// Mitsubishi GX Works2 project: InnerDrumTurnP202201050806   PLC: Q03UDV

PROGRAM MAIN
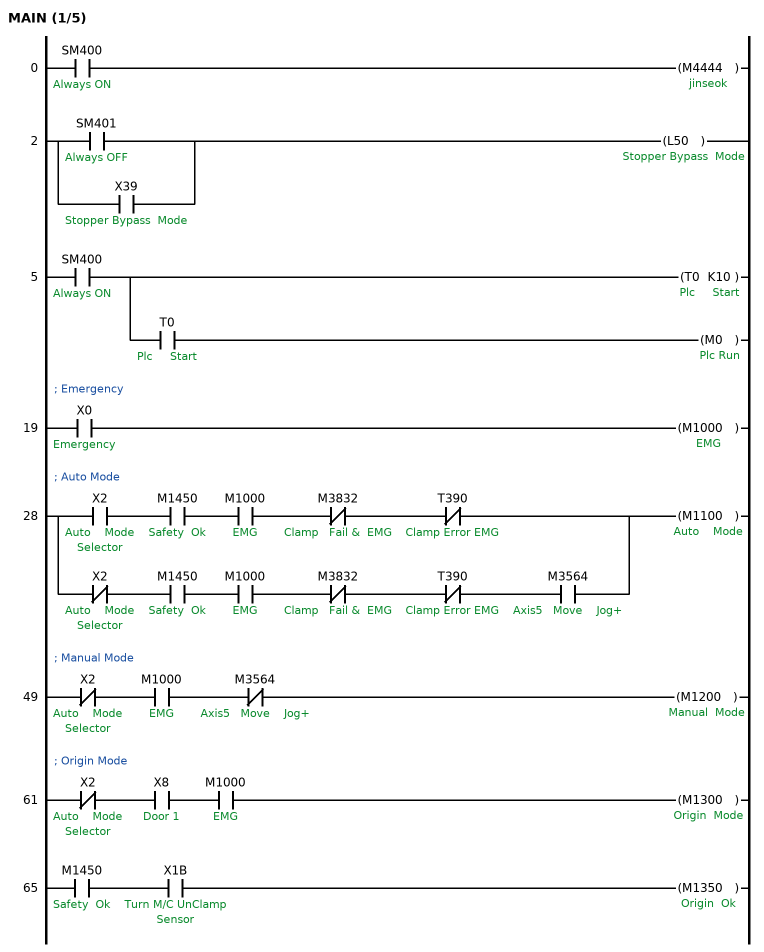
0     LD      SM400  ; Always ON
      OUT     M4444  ; jinseok
2     LD      SM401  ; Always OFF
      OR      X39  ; Stopper Bypass  Mode
      OUT     L50  ; Stopper Bypass  Mode
5     LD      SM400  ; Always ON
      OUT     T0 K10  ; Plc     Start
      AND     T0  ; Plc     Start
      OUT     M0  ; Plc Run
; Emergency
19    LD      X0  ; Emergency
      OUT     M1000  ; EMG
; Auto Mode
28    LD      X2  ; Auto    Mode    Selector
      AND     M1450  ; Safety  Ok
      AND     M1000  ; EMG
      ANI     M3832  ; Clamp   Fail &  EMG
      ANI     T390  ; Clamp Error EMG
      LDI     X2  ; Auto    Mode    Selector
      AND     M1450  ; Safety  Ok
      AND     M1000  ; EMG
      ANI     M3832  ; Clamp   Fail &  EMG
      ANI     T390  ; Clamp Error EMG
      AND     M3564  ; Axis5   Move    Jog+
      ORB
      OUT     M1100  ; Auto    Mode
; Manual Mode
49    LDI     X2  ; Auto    Mode    Selector
      AND     M1000  ; EMG
      ANI     M3564  ; Axis5   Move    Jog+
      OUT     M1200  ; Manual  Mode
; Origin Mode
61    LDI     X2  ; Auto    Mode    Selector
      AND     X8  ; Door 1
      AND     M1000  ; EMG
      OUT     M1300  ; Origin  Mode
65    LD      M1450  ; Safety  Ok
      AND     X1B  ; Turn M/C UnClamp Sensor
      OUT     M1350  ; Origin  Ok
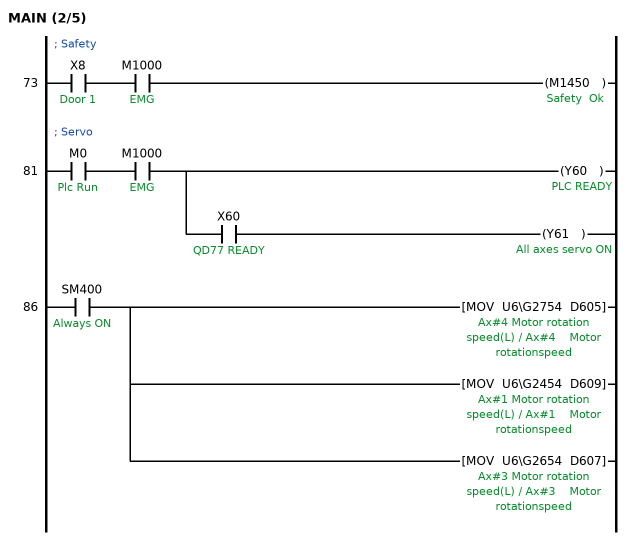
; Safety
73    LD      X8  ; Door 1
      AND     M1000  ; EMG
      OUT     M1450  ; Safety  Ok
; Servo
81    LD      M0  ; Plc Run
      AND     M1000  ; EMG
      OUT     Y60  ; PLC READY
      AND     X60  ; QD77 READY
      OUT     Y61  ; All axes servo ON
86    LD      SM400  ; Always ON
      MOV     U6\G2754 D605  ; Ax#4 Motor rotation speed(L) / Ax#4    Motor   rotationspeed
      MOV     U6\G2454 D609  ; Ax#1 Motor rotation speed(L) / Ax#1    Motor   rotationspeed
      MOV     U6\G2654 D607  ; Ax#3 Motor rotation speed(L) / Ax#3    Motor   rotationspeed
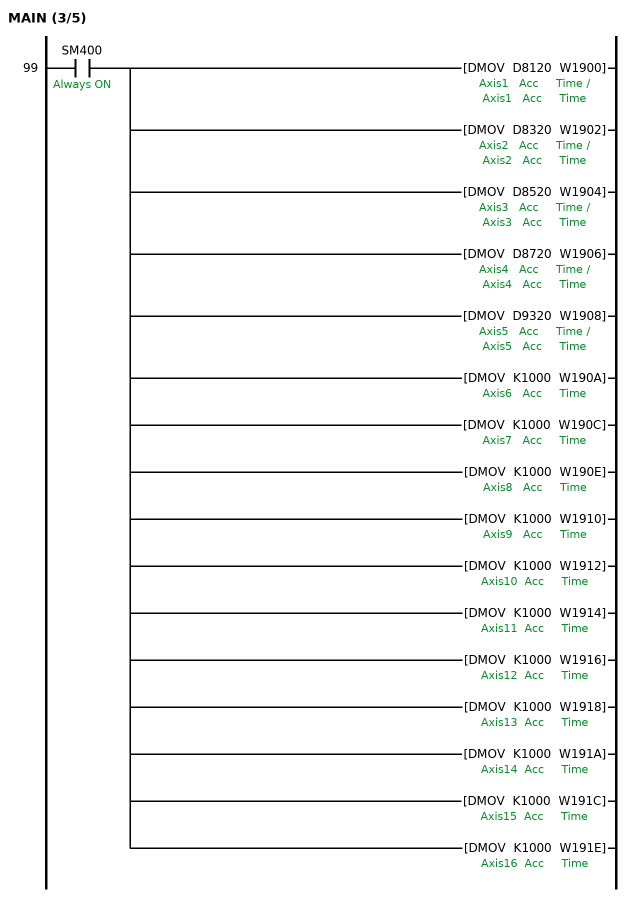
99    LD      SM400  ; Always ON
      DMOV    D8120 W1900  ; Axis1   Acc     Time / Axis1   Acc     Time
      DMOV    D8320 W1902  ; Axis2   Acc     Time / Axis2   Acc     Time
      DMOV    D8520 W1904  ; Axis3   Acc     Time / Axis3   Acc     Time
      DMOV    D8720 W1906  ; Axis4   Acc     Time / Axis4   Acc     Time
      DMOV    D9320 W1908  ; Axis5   Acc     Time / Axis5   Acc     Time
      DMOV    K1000 W190A  ; Axis6   Acc     Time
      DMOV    K1000 W190C  ; Axis7   Acc     Time
      DMOV    K1000 W190E  ; Axis8   Acc     Time
      DMOV    K1000 W1910  ; Axis9   Acc     Time
      DMOV    K1000 W1912  ; Axis10  Acc     Time
      DMOV    K1000 W1914  ; Axis11  Acc     Time
      DMOV    K1000 W1916  ; Axis12  Acc     Time
      DMOV    K1000 W1918  ; Axis13  Acc     Time
      DMOV    K1000 W191A  ; Axis14  Acc     Time
      DMOV    K1000 W191C  ; Axis15  Acc     Time
      DMOV    K1000 W191E  ; Axis16  Acc     Time
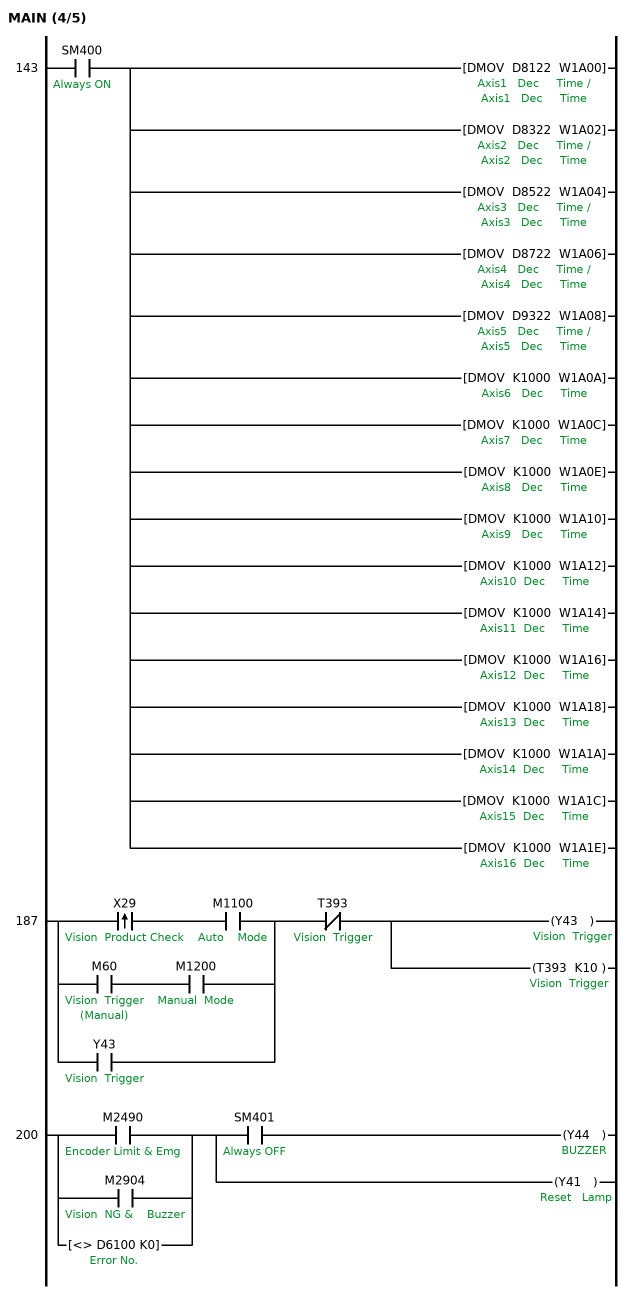
143   LD      SM400  ; Always ON
      DMOV    D8122 W1A00  ; Axis1   Dec     Time / Axis1   Dec     Time
      DMOV    D8322 W1A02  ; Axis2   Dec     Time / Axis2   Dec     Time
      DMOV    D8522 W1A04  ; Axis3   Dec     Time / Axis3   Dec     Time
      DMOV    D8722 W1A06  ; Axis4   Dec     Time / Axis4   Dec     Time
      DMOV    D9322 W1A08  ; Axis5   Dec     Time / Axis5   Dec     Time
      DMOV    K1000 W1A0A  ; Axis6   Dec     Time
      DMOV    K1000 W1A0C  ; Axis7   Dec     Time
      DMOV    K1000 W1A0E  ; Axis8   Dec     Time
      DMOV    K1000 W1A10  ; Axis9   Dec     Time
      DMOV    K1000 W1A12  ; Axis10  Dec     Time
      DMOV    K1000 W1A14  ; Axis11  Dec     Time
      DMOV    K1000 W1A16  ; Axis12  Dec     Time
      DMOV    K1000 W1A18  ; Axis13  Dec     Time
      DMOV    K1000 W1A1A  ; Axis14  Dec     Time
      DMOV    K1000 W1A1C  ; Axis15  Dec     Time
      DMOV    K1000 W1A1E  ; Axis16  Dec     Time
187   LDP     X29  ; Vision  Product Check
      AND     M1100  ; Auto    Mode
      LD      M60  ; Vision  Trigger (Manual)
      AND     M1200  ; Manual  Mode
      ORB
      OR      Y43  ; Vision  Trigger
      ANI     T393  ; Vision  Trigger
      OUT     Y43  ; Vision  Trigger
      OUT     T393 K10  ; Vision  Trigger
200   LD      M2490  ; Encoder Limit & Emg
      OR      M2904  ; Vision  NG &    Buzzer
      OR<>    D6100 K0  ; Error No.
      MPS
      AND     SM401  ; Always OFF
      OUT     Y44  ; BUZZER
      MPP
      OUT     Y41  ; Reset   Lamp
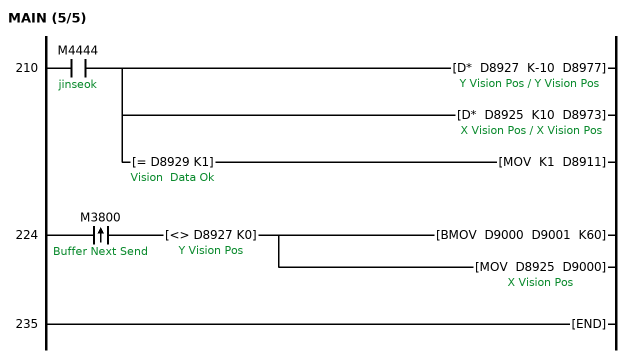
210   LD      M4444  ; jinseok
      D*      D8927 K-10 D8977  ; Y Vision Pos / Y Vision Pos
      D*      D8925 K10 D8973  ; X Vision Pos / X Vision Pos
      AND=    D8929 K1  ; Vision  Data Ok
      MOV     K1 D8911
224   LDP     M3800  ; Buffer Next Send
      AND<>   D8927 K0  ; Y Vision Pos
      BMOV    D9000 D9001 K60
      MOV     D8925 D9000
235   END
END_PROGRAM

PROGRAM AUTO
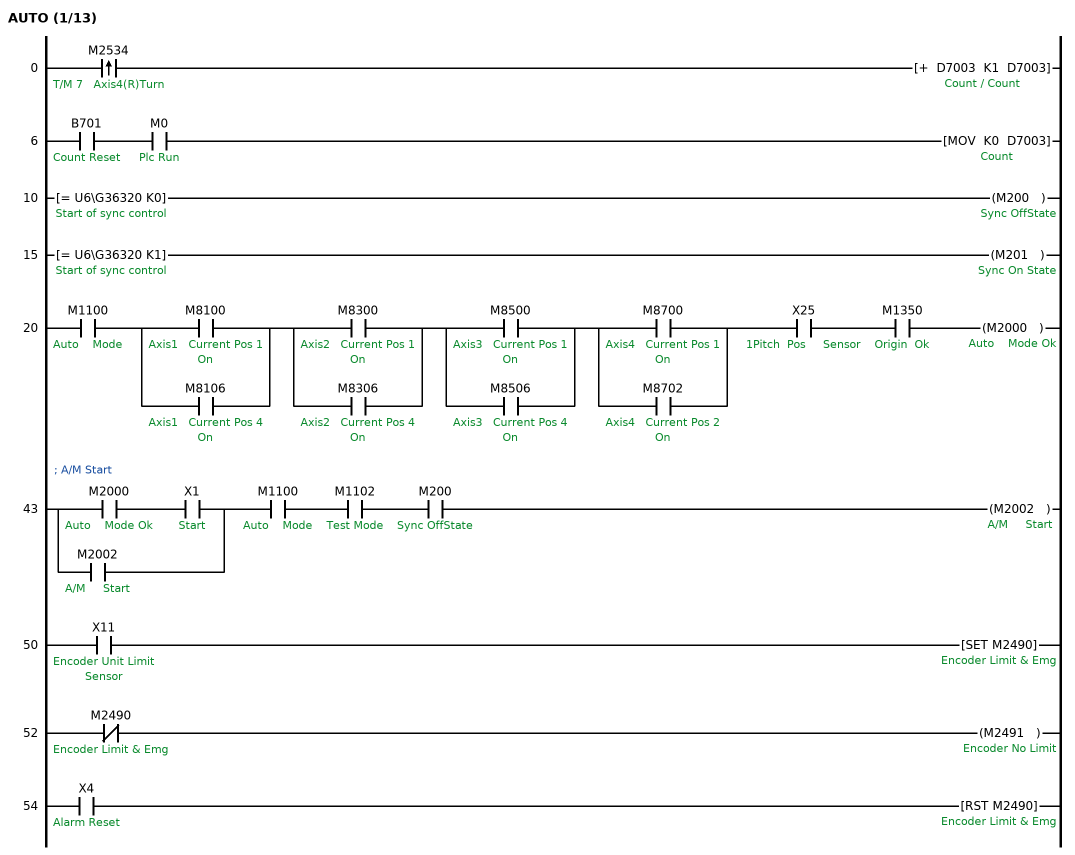
0     LDP     M2534  ; T/M 7   Axis4(R)Turn
      +       D7003 K1 D7003  ; Count
6     LD      B701  ; Count Reset
      AND     M0  ; Plc Run
      MOV     K0 D7003
10    LD=     U6\G36320 K0  ; Start of sync control
      OUT     M200  ; Sync OffState
15    LD=     U6\G36320 K1  ; Start of sync control
      OUT     M201  ; Sync On State
20    LD      M1100  ; Auto    Mode
      LD      M8100  ; Axis1   Current Pos 1 On
      OR      M8106  ; Axis1   Current Pos 4 On
      ANB
      LD      M8300  ; Axis2   Current Pos 1 On
      OR      M8306  ; Axis2   Current Pos 4 On
      ANB
      LD      M8500  ; Axis3   Current Pos 1 On
      OR      M8506  ; Axis3   Current Pos 4 On
      ANB
      LD      M8700  ; Axis4   Current Pos 1 On
      OR      M8702  ; Axis4   Current Pos 2 On
      ANB
      AND     X25  ; 1Pitch  Pos     Sensor
      AND     M1350  ; Origin  Ok
      OUT     M2000  ; Auto    Mode Ok
; A/M Start
43    LD      M2000  ; Auto    Mode Ok
      AND     X1  ; Start
      OR      M2002  ; A/M     Start
      AND     M1100  ; Auto    Mode
      AND     M1102  ; Test Mode
      AND     M200  ; Sync OffState
      OUT     M2002  ; A/M     Start
50    LD      X11  ; Encoder Unit Limit Sensor
      SET     M2490  ; Encoder Limit & Emg
52    LDI     M2490  ; Encoder Limit & Emg
      OUT     M2491  ; Encoder No Limit
54    LD      X4  ; Alarm Reset
      RST     M2490  ; Encoder Limit & Emg
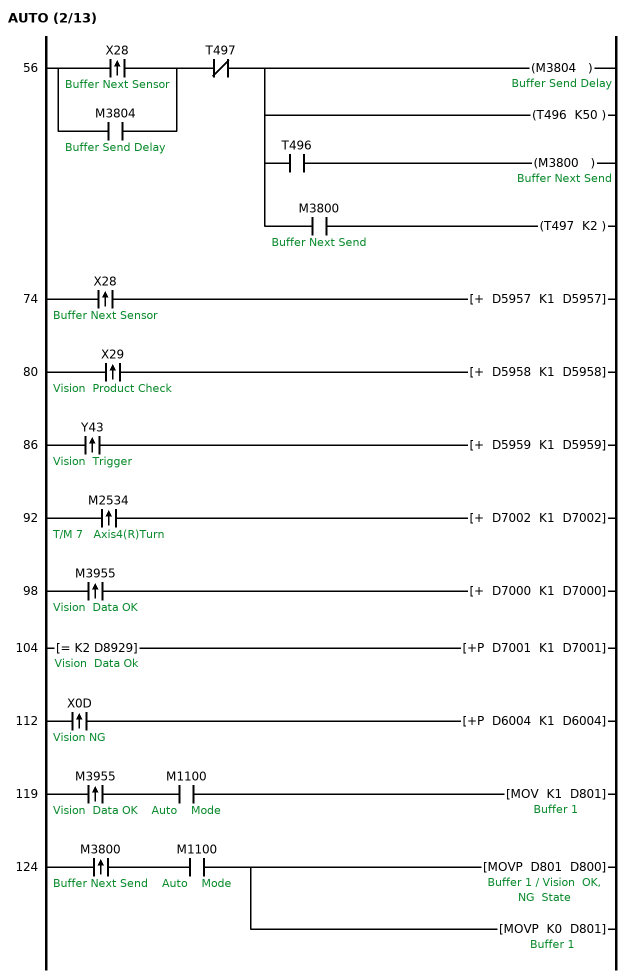
56    LDP     X28  ; Buffer Next Sensor
      OR      M3804  ; Buffer Send Delay
      ANI     T497
      OUT     M3804  ; Buffer Send Delay
      OUT     T496 K50
      MPS
      AND     T496
      OUT     M3800  ; Buffer Next Send
      MPP
      AND     M3800  ; Buffer Next Send
      OUT     T497 K2
74    LDP     X28  ; Buffer Next Sensor
      +       D5957 K1 D5957
80    LDP     X29  ; Vision  Product Check
      +       D5958 K1 D5958
86    LDP     Y43  ; Vision  Trigger
      +       D5959 K1 D5959
92    LDP     M2534  ; T/M 7   Axis4(R)Turn
      +       D7002 K1 D7002
98    LDP     M3955  ; Vision  Data OK
      +       D7000 K1 D7000
104   LD=     K2 D8929  ; Vision  Data Ok
      +P      D7001 K1 D7001
112   LDP     X0D  ; Vision NG
      +P      D6004 K1 D6004
119   LDP     M3955  ; Vision  Data OK
      AND     M1100  ; Auto    Mode
      MOV     K1 D801  ; Buffer 1
124   LDP     M3800  ; Buffer Next Send
      AND     M1100  ; Auto    Mode
      MOVP    D801 D800  ; Vision  OK, NG  State
      MOVP    K0 D801
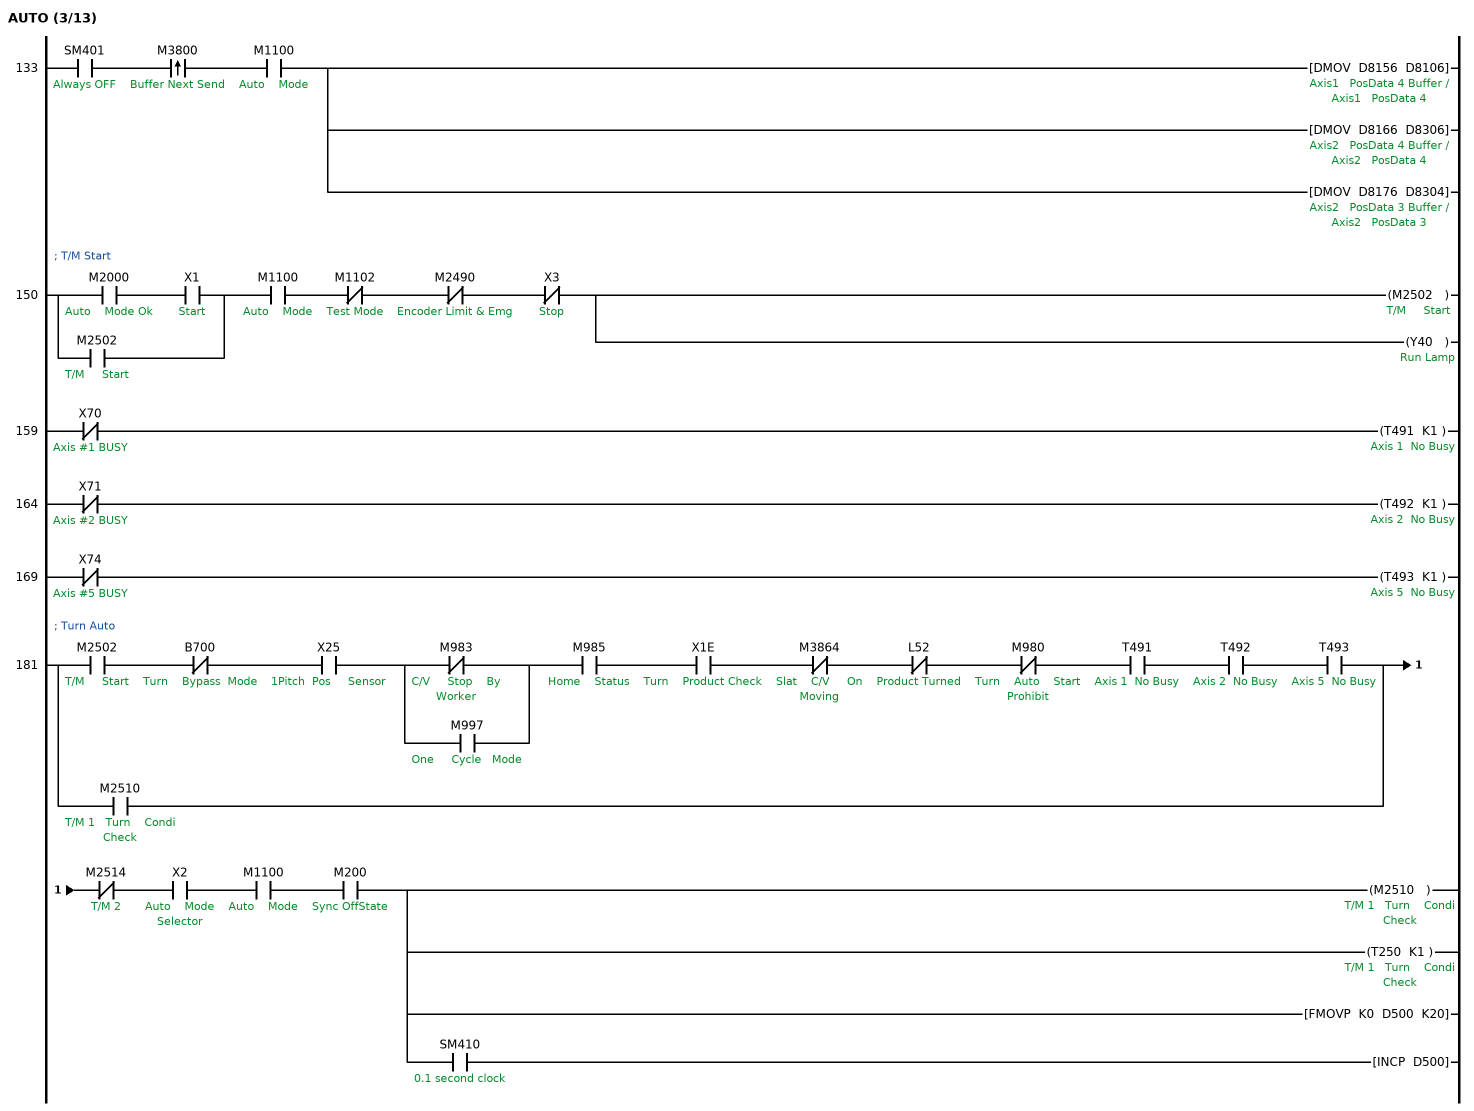
133   LD      SM401  ; Always OFF
      ANDP    M3800  ; Buffer Next Send
      AND     M1100  ; Auto    Mode
      DMOV    D8156 D8106  ; Axis1   PosData 4 Buffer / Axis1   PosData 4
      DMOV    D8166 D8306  ; Axis2   PosData 4 Buffer / Axis2   PosData 4
      DMOV    D8176 D8304  ; Axis2   PosData 3 Buffer / Axis2   PosData 3
; T/M Start
150   LD      M2000  ; Auto    Mode Ok
      AND     X1  ; Start
      OR      M2502  ; T/M     Start
      AND     M1100  ; Auto    Mode
      ANI     M1102  ; Test Mode
      ANI     M2490  ; Encoder Limit & Emg
      ANI     X3  ; Stop
      OUT     M2502  ; T/M     Start
      OUT     Y40  ; Run Lamp
159   LDI     X70  ; Axis #1 BUSY
      OUT     T491 K1  ; Axis 1  No Busy
164   LDI     X71  ; Axis #2 BUSY
      OUT     T492 K1  ; Axis 2  No Busy
169   LDI     X74  ; Axis #5 BUSY
      OUT     T493 K1  ; Axis 5  No Busy
; Turn Auto
181   LD      M2502  ; T/M     Start
      ANI     B700  ; Turn    Bypass  Mode
      AND     X25  ; 1Pitch  Pos     Sensor
      LDI     M983  ; C/V     Stop    By      Worker
      OR      M997  ; One     Cycle   Mode
      ANB
      AND     M985  ; Home    Status
      AND     X1E  ; Turn    Product Check
      ANI     M3864  ; Slat    C/V     On      Moving
      ANI     L52  ; Product Turned
      ANI     M980  ; Turn    Auto    Start   Prohibit
      AND     T491  ; Axis 1  No Busy
      AND     T492  ; Axis 2  No Busy
      AND     T493  ; Axis 5  No Busy
      OR      M2510  ; T/M 1   Turn    Condi   Check
      ANI     M2514  ; T/M 2
      AND     X2  ; Auto    Mode    Selector
      AND     M1100  ; Auto    Mode
      AND     M200  ; Sync OffState
      OUT     M2510  ; T/M 1   Turn    Condi   Check
      OUT     T250 K1  ; T/M 1   Turn    Condi   Check
      FMOVP   K0 D500 K20
      AND     SM410  ; 0.1 second clock
      INCP    D500
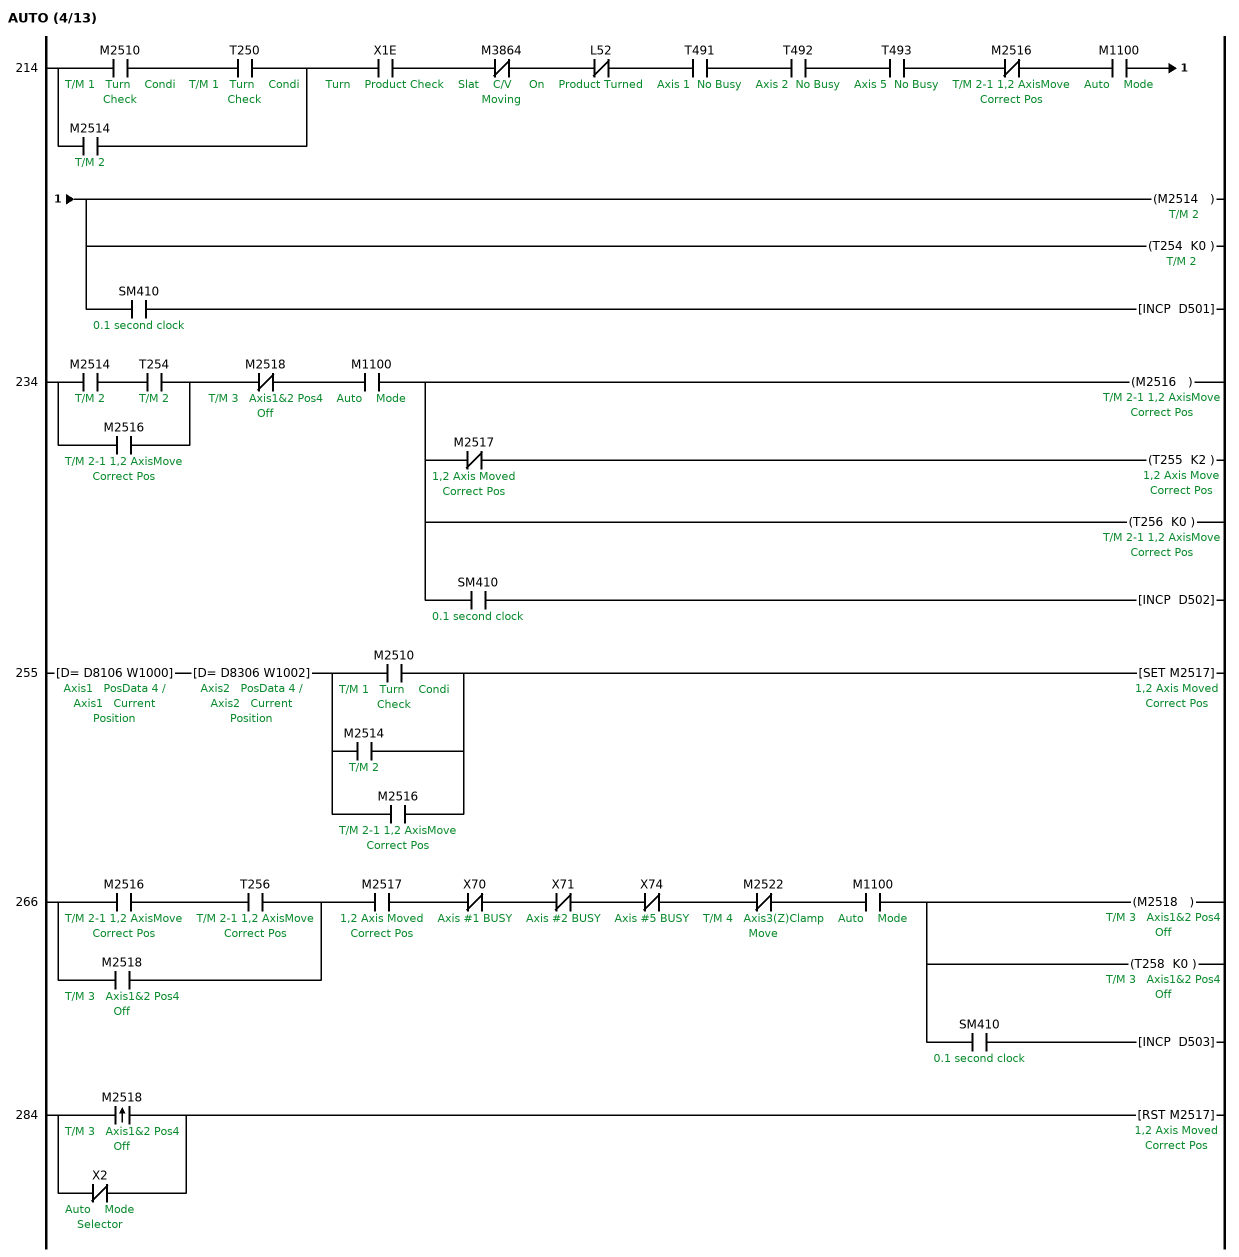
214   LD      M2510  ; T/M 1   Turn    Condi   Check
      AND     T250  ; T/M 1   Turn    Condi   Check
      OR      M2514  ; T/M 2
      AND     X1E  ; Turn    Product Check
      ANI     M3864  ; Slat    C/V     On      Moving
      ANI     L52  ; Product Turned
      AND     T491  ; Axis 1  No Busy
      AND     T492  ; Axis 2  No Busy
      AND     T493  ; Axis 5  No Busy
      ANI     M2516  ; T/M 2-1 1,2 AxisMove Correct Pos
      AND     M1100  ; Auto    Mode
      OUT     M2514  ; T/M 2
      OUT     T254 K0  ; T/M 2
      AND     SM410  ; 0.1 second clock
      INCP    D501
234   LD      M2514  ; T/M 2
      AND     T254  ; T/M 2
      OR      M2516  ; T/M 2-1 1,2 AxisMove Correct Pos
      ANI     M2518  ; T/M 3   Axis1&2 Pos4    Off
      AND     M1100  ; Auto    Mode
      OUT     M2516  ; T/M 2-1 1,2 AxisMove Correct Pos
      MPS
      ANI     M2517  ; 1,2 Axis Moved Correct Pos
      OUT     T255 K2  ; 1,2 Axis Move Correct Pos
      MPP
      OUT     T256 K0  ; T/M 2-1 1,2 AxisMove Correct Pos
      AND     SM410  ; 0.1 second clock
      INCP    D502
255   LDD=    D8106 W1000  ; Axis1   PosData 4 / Axis1   Current Position
      ANDD=   D8306 W1002  ; Axis2   PosData 4 / Axis2   Current Position
      LD      M2510  ; T/M 1   Turn    Condi   Check
      OR      M2514  ; T/M 2
      OR      M2516  ; T/M 2-1 1,2 AxisMove Correct Pos
      ANB
      SET     M2517  ; 1,2 Axis Moved Correct Pos
266   LD      M2516  ; T/M 2-1 1,2 AxisMove Correct Pos
      AND     T256  ; T/M 2-1 1,2 AxisMove Correct Pos
      OR      M2518  ; T/M 3   Axis1&2 Pos4    Off
      AND     M2517  ; 1,2 Axis Moved Correct Pos
      ANI     X70  ; Axis #1 BUSY
      ANI     X71  ; Axis #2 BUSY
      ANI     X74  ; Axis #5 BUSY
      ANI     M2522  ; T/M 4   Axis3(Z)Clamp   Move
      AND     M1100  ; Auto    Mode
      OUT     M2518  ; T/M 3   Axis1&2 Pos4    Off
      OUT     T258 K0  ; T/M 3   Axis1&2 Pos4    Off
      AND     SM410  ; 0.1 second clock
      INCP    D503
284   LDP     M2518  ; T/M 3   Axis1&2 Pos4    Off
      ORI     X2  ; Auto    Mode    Selector
      RST     M2517  ; 1,2 Axis Moved Correct Pos
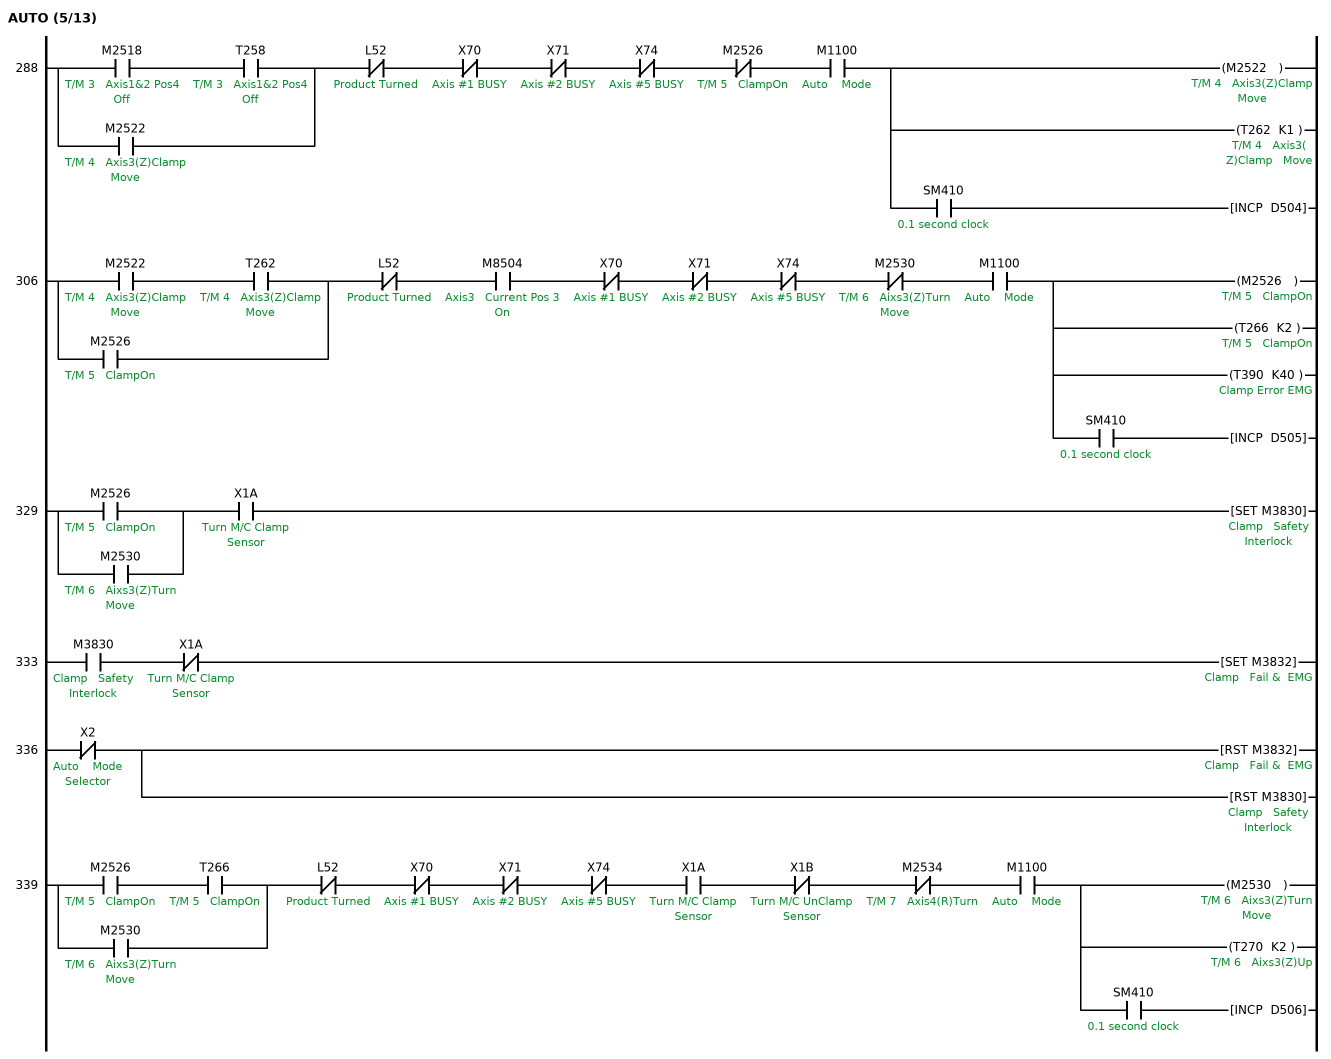
288   LD      M2518  ; T/M 3   Axis1&2 Pos4    Off
      AND     T258  ; T/M 3   Axis1&2 Pos4    Off
      OR      M2522  ; T/M 4   Axis3(Z)Clamp   Move
      ANI     L52  ; Product Turned
      ANI     X70  ; Axis #1 BUSY
      ANI     X71  ; Axis #2 BUSY
      ANI     X74  ; Axis #5 BUSY
      ANI     M2526  ; T/M 5   ClampOn
      AND     M1100  ; Auto    Mode
      OUT     M2522  ; T/M 4   Axis3(Z)Clamp   Move
      OUT     T262 K1  ; T/M 4   Axis3(Z)Clamp   Move
      AND     SM410  ; 0.1 second clock
      INCP    D504
306   LD      M2522  ; T/M 4   Axis3(Z)Clamp   Move
      AND     T262  ; T/M 4   Axis3(Z)Clamp   Move
      OR      M2526  ; T/M 5   ClampOn
      ANI     L52  ; Product Turned
      AND     M8504  ; Axis3   Current Pos 3 On
      ANI     X70  ; Axis #1 BUSY
      ANI     X71  ; Axis #2 BUSY
      ANI     X74  ; Axis #5 BUSY
      ANI     M2530  ; T/M 6   Aixs3(Z)Turn    Move
      AND     M1100  ; Auto    Mode
      OUT     M2526  ; T/M 5   ClampOn
      OUT     T266 K2  ; T/M 5   ClampOn
      OUT     T390 K40  ; Clamp Error EMG
      AND     SM410  ; 0.1 second clock
      INCP    D505
329   LD      M2526  ; T/M 5   ClampOn
      OR      M2530  ; T/M 6   Aixs3(Z)Turn    Move
      AND     X1A  ; Turn M/C Clamp Sensor
      SET     M3830  ; Clamp   Safety  Interlock
333   LD      M3830  ; Clamp   Safety  Interlock
      ANI     X1A  ; Turn M/C Clamp Sensor
      SET     M3832  ; Clamp   Fail &  EMG
336   LDI     X2  ; Auto    Mode    Selector
      RST     M3832  ; Clamp   Fail &  EMG
      RST     M3830  ; Clamp   Safety  Interlock
339   LD      M2526  ; T/M 5   ClampOn
      AND     T266  ; T/M 5   ClampOn
      OR      M2530  ; T/M 6   Aixs3(Z)Turn    Move
      ANI     L52  ; Product Turned
      ANI     X70  ; Axis #1 BUSY
      ANI     X71  ; Axis #2 BUSY
      ANI     X74  ; Axis #5 BUSY
      AND     X1A  ; Turn M/C Clamp Sensor
      ANI     X1B  ; Turn M/C UnClamp Sensor
      ANI     M2534  ; T/M 7   Axis4(R)Turn
      AND     M1100  ; Auto    Mode
      OUT     M2530  ; T/M 6   Aixs3(Z)Turn    Move
      OUT     T270 K2  ; T/M 6   Aixs3(Z)Up
      AND     SM410  ; 0.1 second clock
      INCP    D506
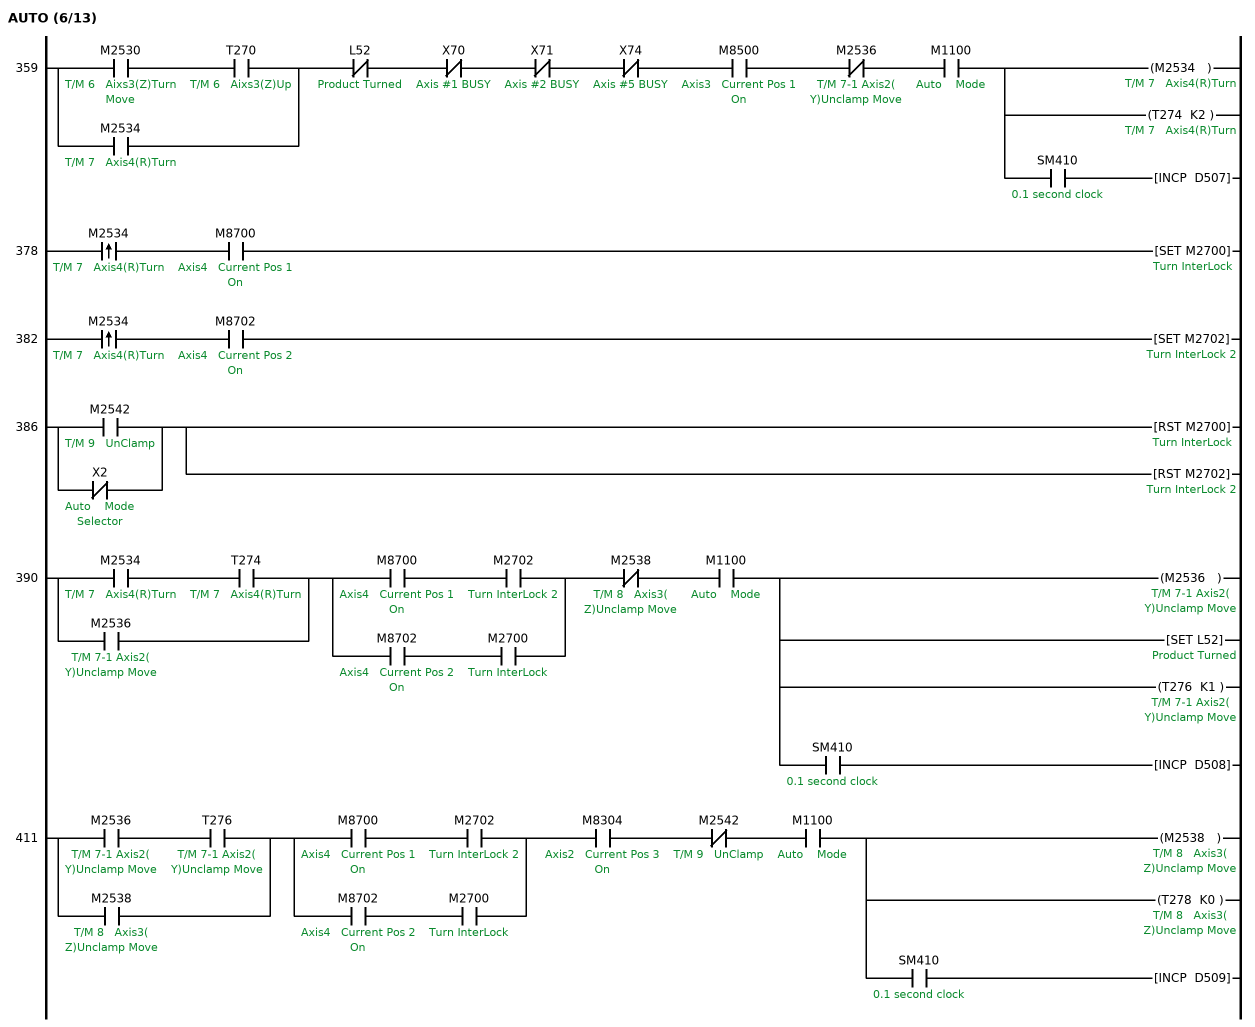
359   LD      M2530  ; T/M 6   Aixs3(Z)Turn    Move
      AND     T270  ; T/M 6   Aixs3(Z)Up
      OR      M2534  ; T/M 7   Axis4(R)Turn
      ANI     L52  ; Product Turned
      ANI     X70  ; Axis #1 BUSY
      ANI     X71  ; Axis #2 BUSY
      ANI     X74  ; Axis #5 BUSY
      AND     M8500  ; Axis3   Current Pos 1 On
      ANI     M2536  ; T/M 7-1 Axis2(Y)Unclamp Move
      AND     M1100  ; Auto    Mode
      OUT     M2534  ; T/M 7   Axis4(R)Turn
      OUT     T274 K2  ; T/M 7   Axis4(R)Turn
      AND     SM410  ; 0.1 second clock
      INCP    D507
378   LDP     M2534  ; T/M 7   Axis4(R)Turn
      AND     M8700  ; Axis4   Current Pos 1 On
      SET     M2700  ; Turn InterLock
382   LDP     M2534  ; T/M 7   Axis4(R)Turn
      AND     M8702  ; Axis4   Current Pos 2 On
      SET     M2702  ; Turn InterLock 2
386   LD      M2542  ; T/M 9   UnClamp
      ORI     X2  ; Auto    Mode    Selector
      RST     M2700  ; Turn InterLock
      RST     M2702  ; Turn InterLock 2
390   LD      M2534  ; T/M 7   Axis4(R)Turn
      AND     T274  ; T/M 7   Axis4(R)Turn
      OR      M2536  ; T/M 7-1 Axis2(Y)Unclamp Move
      LD      M8700  ; Axis4   Current Pos 1 On
      AND     M2702  ; Turn InterLock 2
      LD      M8702  ; Axis4   Current Pos 2 On
      AND     M2700  ; Turn InterLock
      ORB
      ANB
      ANI     M2538  ; T/M 8   Axis3(Z)Unclamp Move
      AND     M1100  ; Auto    Mode
      OUT     M2536  ; T/M 7-1 Axis2(Y)Unclamp Move
      SET     L52  ; Product Turned
      OUT     T276 K1  ; T/M 7-1 Axis2(Y)Unclamp Move
      AND     SM410  ; 0.1 second clock
      INCP    D508
411   LD      M2536  ; T/M 7-1 Axis2(Y)Unclamp Move
      AND     T276  ; T/M 7-1 Axis2(Y)Unclamp Move
      OR      M2538  ; T/M 8   Axis3(Z)Unclamp Move
      LD      M8700  ; Axis4   Current Pos 1 On
      AND     M2702  ; Turn InterLock 2
      LD      M8702  ; Axis4   Current Pos 2 On
      AND     M2700  ; Turn InterLock
      ORB
      ANB
      AND     M8304  ; Axis2   Current Pos 3 On
      ANI     M2542  ; T/M 9   UnClamp
      AND     M1100  ; Auto    Mode
      OUT     M2538  ; T/M 8   Axis3(Z)Unclamp Move
      OUT     T278 K0  ; T/M 8   Axis3(Z)Unclamp Move
      AND     SM410  ; 0.1 second clock
      INCP    D509
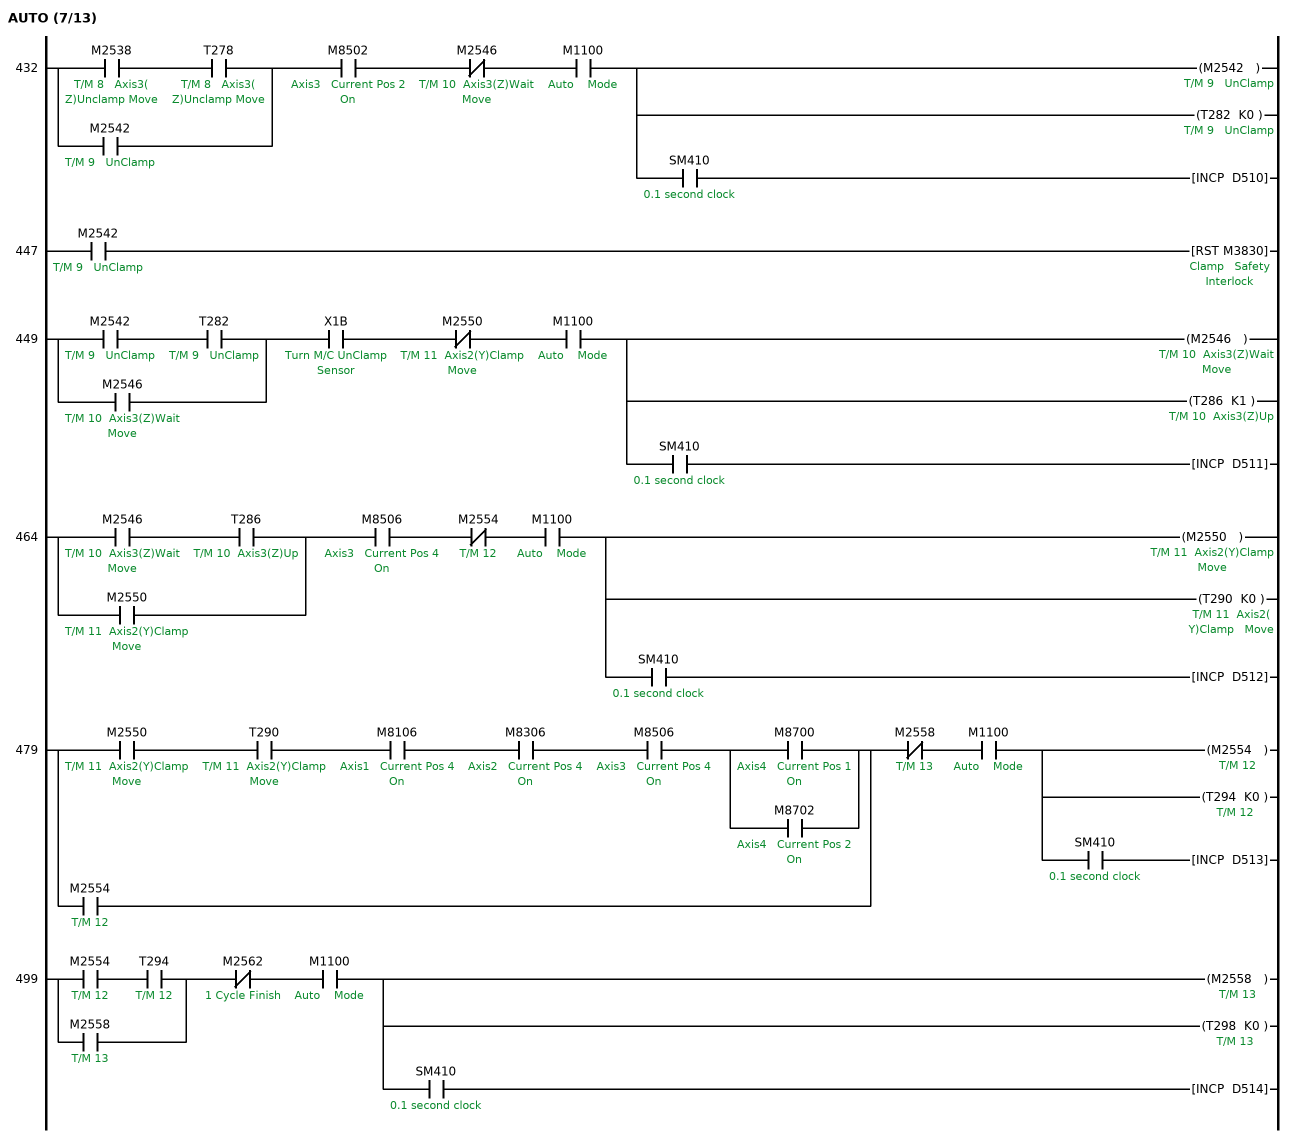
432   LD      M2538  ; T/M 8   Axis3(Z)Unclamp Move
      AND     T278  ; T/M 8   Axis3(Z)Unclamp Move
      OR      M2542  ; T/M 9   UnClamp
      AND     M8502  ; Axis3   Current Pos 2 On
      ANI     M2546  ; T/M 10  Axis3(Z)Wait    Move
      AND     M1100  ; Auto    Mode
      OUT     M2542  ; T/M 9   UnClamp
      OUT     T282 K0  ; T/M 9   UnClamp
      AND     SM410  ; 0.1 second clock
      INCP    D510
447   LD      M2542  ; T/M 9   UnClamp
      RST     M3830  ; Clamp   Safety  Interlock
449   LD      M2542  ; T/M 9   UnClamp
      AND     T282  ; T/M 9   UnClamp
      OR      M2546  ; T/M 10  Axis3(Z)Wait    Move
      AND     X1B  ; Turn M/C UnClamp Sensor
      ANI     M2550  ; T/M 11  Axis2(Y)Clamp   Move
      AND     M1100  ; Auto    Mode
      OUT     M2546  ; T/M 10  Axis3(Z)Wait    Move
      OUT     T286 K1  ; T/M 10  Axis3(Z)Up
      AND     SM410  ; 0.1 second clock
      INCP    D511
464   LD      M2546  ; T/M 10  Axis3(Z)Wait    Move
      AND     T286  ; T/M 10  Axis3(Z)Up
      OR      M2550  ; T/M 11  Axis2(Y)Clamp   Move
      AND     M8506  ; Axis3   Current Pos 4 On
      ANI     M2554  ; T/M 12
      AND     M1100  ; Auto    Mode
      OUT     M2550  ; T/M 11  Axis2(Y)Clamp   Move
      OUT     T290 K0  ; T/M 11  Axis2(Y)Clamp   Move
      AND     SM410  ; 0.1 second clock
      INCP    D512
479   LD      M2550  ; T/M 11  Axis2(Y)Clamp   Move
      AND     T290  ; T/M 11  Axis2(Y)Clamp   Move
      AND     M8106  ; Axis1   Current Pos 4 On
      AND     M8306  ; Axis2   Current Pos 4 On
      AND     M8506  ; Axis3   Current Pos 4 On
      LD      M8700  ; Axis4   Current Pos 1 On
      OR      M8702  ; Axis4   Current Pos 2 On
      ANB
      OR      M2554  ; T/M 12
      ANI     M2558  ; T/M 13
      AND     M1100  ; Auto    Mode
      OUT     M2554  ; T/M 12
      OUT     T294 K0  ; T/M 12
      AND     SM410  ; 0.1 second clock
      INCP    D513
499   LD      M2554  ; T/M 12
      AND     T294  ; T/M 12
      OR      M2558  ; T/M 13
      ANI     M2562  ; 1 Cycle Finish
      AND     M1100  ; Auto    Mode
      OUT     M2558  ; T/M 13
      OUT     T298 K0  ; T/M 13
      AND     SM410  ; 0.1 second clock
      INCP    D514
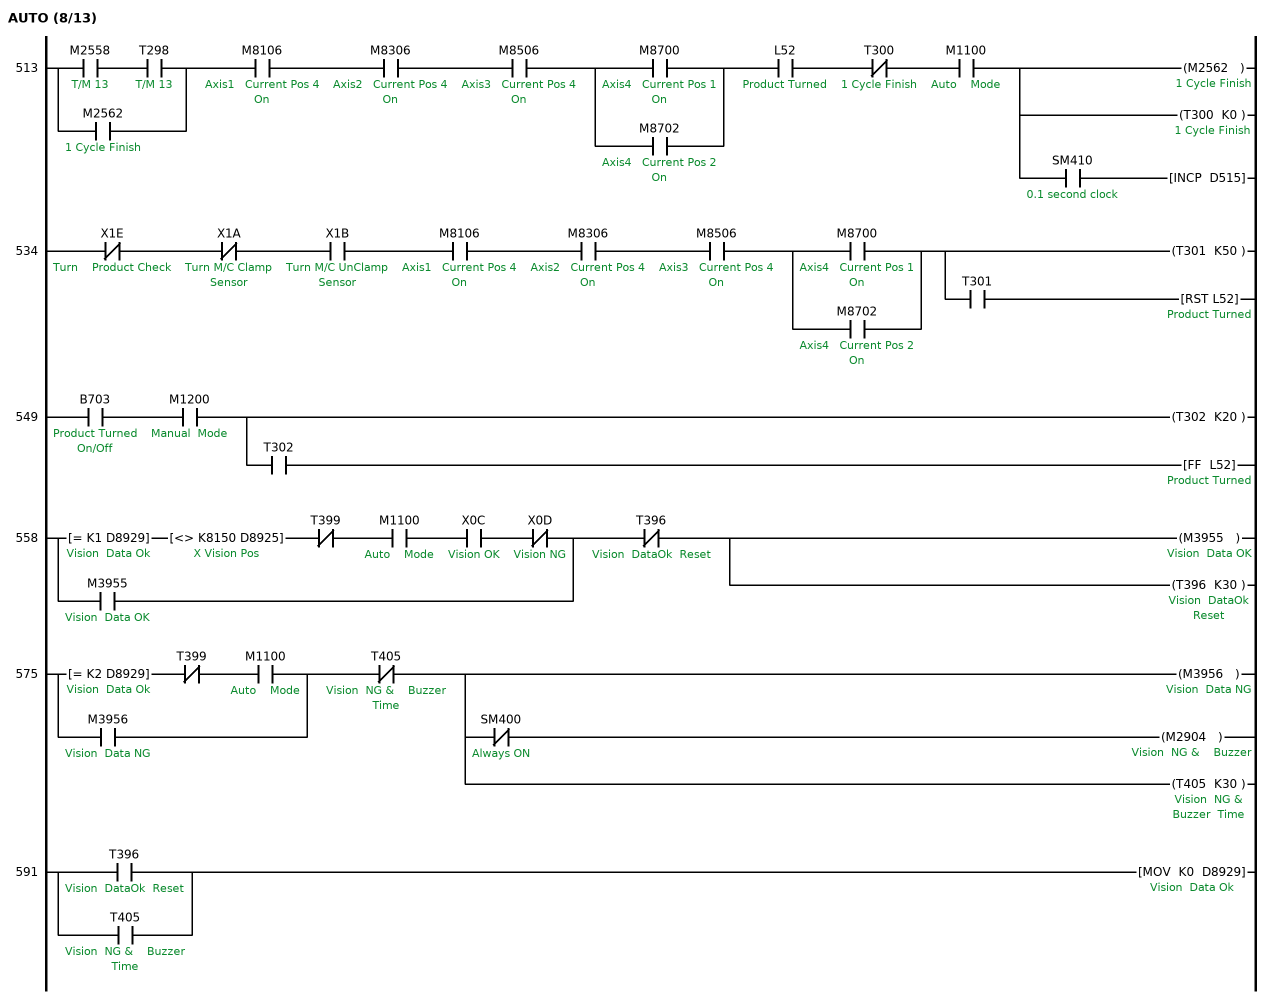
513   LD      M2558  ; T/M 13
      AND     T298  ; T/M 13
      OR      M2562  ; 1 Cycle Finish
      AND     M8106  ; Axis1   Current Pos 4 On
      AND     M8306  ; Axis2   Current Pos 4 On
      AND     M8506  ; Axis3   Current Pos 4 On
      LD      M8700  ; Axis4   Current Pos 1 On
      OR      M8702  ; Axis4   Current Pos 2 On
      ANB
      AND     L52  ; Product Turned
      ANI     T300  ; 1 Cycle Finish
      AND     M1100  ; Auto    Mode
      OUT     M2562  ; 1 Cycle Finish
      OUT     T300 K0  ; 1 Cycle Finish
      AND     SM410  ; 0.1 second clock
      INCP    D515
534   LDI     X1E  ; Turn    Product Check
      ANI     X1A  ; Turn M/C Clamp Sensor
      AND     X1B  ; Turn M/C UnClamp Sensor
      AND     M8106  ; Axis1   Current Pos 4 On
      AND     M8306  ; Axis2   Current Pos 4 On
      AND     M8506  ; Axis3   Current Pos 4 On
      LD      M8700  ; Axis4   Current Pos 1 On
      OR      M8702  ; Axis4   Current Pos 2 On
      ANB
      OUT     T301 K50
      AND     T301
      RST     L52  ; Product Turned
549   LD      B703  ; Product Turned  On/Off
      AND     M1200  ; Manual  Mode
      OUT     T302 K20
      AND     T302
      FF      L52
558   LD=     K1 D8929  ; Vision  Data Ok
      AND<>   K8150 D8925  ; X Vision Pos
      ANI     T399
      AND     M1100  ; Auto    Mode
      AND     X0C  ; Vision OK
      ANI     X0D  ; Vision NG
      OR      M3955  ; Vision  Data OK
      ANI     T396  ; Vision  DataOk  Reset
      OUT     M3955  ; Vision  Data OK
      OUT     T396 K30  ; Vision  DataOk  Reset
575   LD=     K2 D8929  ; Vision  Data Ok
      ANI     T399
      AND     M1100  ; Auto    Mode
      OR      M3956  ; Vision  Data NG
      ANI     T405  ; Vision  NG &    Buzzer  Time
      OUT     M3956  ; Vision  Data NG
      MPS
      ANI     SM400  ; Always ON
      OUT     M2904  ; Vision  NG &    Buzzer
      MPP
      OUT     T405 K30  ; Vision  NG &    Buzzer  Time
591   LD      T396  ; Vision  DataOk  Reset
      OR      T405  ; Vision  NG &    Buzzer  Time
      MOV     K0 D8929
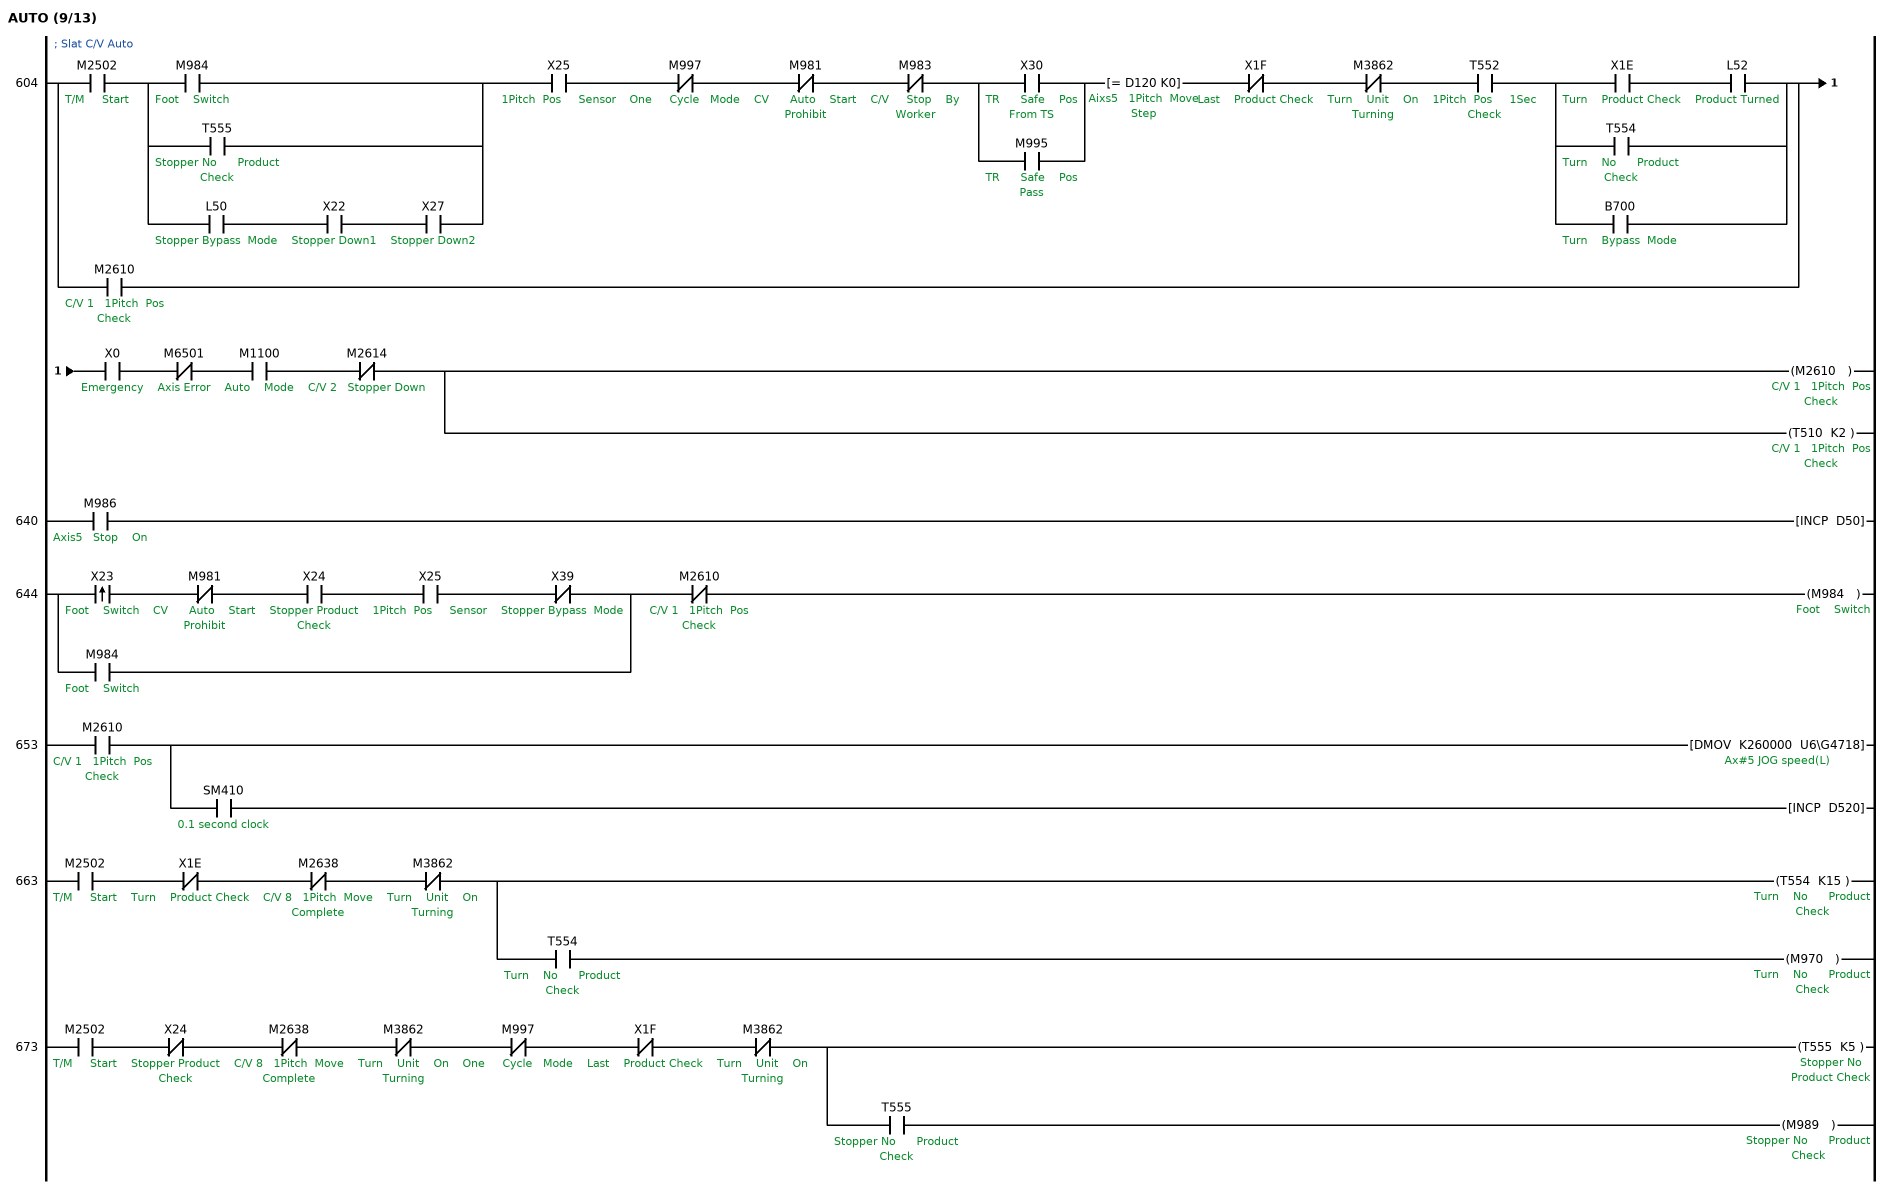
; Slat C/V Auto
604   LD      M2502  ; T/M     Start
      LD      M984  ; Foot    Switch
      OR      T555  ; Stopper No      Product Check
      LD      L50  ; Stopper Bypass  Mode
      AND     X22  ; Stopper Down1
      AND     X27  ; Stopper Down2
      ORB
      ANB
      AND     X25  ; 1Pitch  Pos     Sensor
      ANI     M997  ; One     Cycle   Mode
      ANI     M981  ; CV      Auto    Start   Prohibit
      ANI     M983  ; C/V     Stop    By      Worker
      LD      X30  ; TR      Safe    Pos     From TS
      OR      M995  ; TR      Safe    Pos     Pass
      ANB
      AND=    D120 K0  ; Aixs5   1Pitch  Move    Step
      ANI     X1F  ; Last    Product Check
      ANI     M3862  ; Turn    Unit    On      Turning
      AND     T552  ; 1Pitch  Pos     1Sec    Check
      LD      X1E  ; Turn    Product Check
      AND     L52  ; Product Turned
      OR      T554  ; Turn    No      Product Check
      OR      B700  ; Turn    Bypass  Mode
      ANB
      OR      M2610  ; C/V 1   1Pitch  Pos     Check
      AND     X0  ; Emergency
      ANI     M6501  ; Axis Error
      AND     M1100  ; Auto    Mode
      ANI     M2614  ; C/V 2   Stopper Down
      OUT     M2610  ; C/V 1   1Pitch  Pos     Check
      OUT     T510 K2  ; C/V 1   1Pitch  Pos     Check
640   LD      M986  ; Axis5   Stop    On
      INCP    D50
644   LDP     X23  ; Foot    Switch
      ANI     M981  ; CV      Auto    Start   Prohibit
      AND     X24  ; Stopper Product Check
      AND     X25  ; 1Pitch  Pos     Sensor
      ANI     X39  ; Stopper Bypass  Mode
      OR      M984  ; Foot    Switch
      ANI     M2610  ; C/V 1   1Pitch  Pos     Check
      OUT     M984  ; Foot    Switch
653   LD      M2610  ; C/V 1   1Pitch  Pos     Check
      DMOV    K260000 U6\G4718  ; Ax#5 JOG speed(L)
      AND     SM410  ; 0.1 second clock
      INCP    D520
663   LD      M2502  ; T/M     Start
      ANI     X1E  ; Turn    Product Check
      ANI     M2638  ; C/V 8   1Pitch  Move    Complete
      ANI     M3862  ; Turn    Unit    On      Turning
      OUT     T554 K15  ; Turn    No      Product Check
      AND     T554  ; Turn    No      Product Check
      OUT     M970  ; Turn    No      Product Check
673   LD      M2502  ; T/M     Start
      ANI     X24  ; Stopper Product Check
      ANI     M2638  ; C/V 8   1Pitch  Move    Complete
      ANI     M3862  ; Turn    Unit    On      Turning
      ANI     M997  ; One     Cycle   Mode
      ANI     X1F  ; Last    Product Check
      ANI     M3862  ; Turn    Unit    On      Turning
      OUT     T555 K5  ; Stopper No      Product Check
      AND     T555  ; Stopper No      Product Check
      OUT     M989  ; Stopper No      Product Check
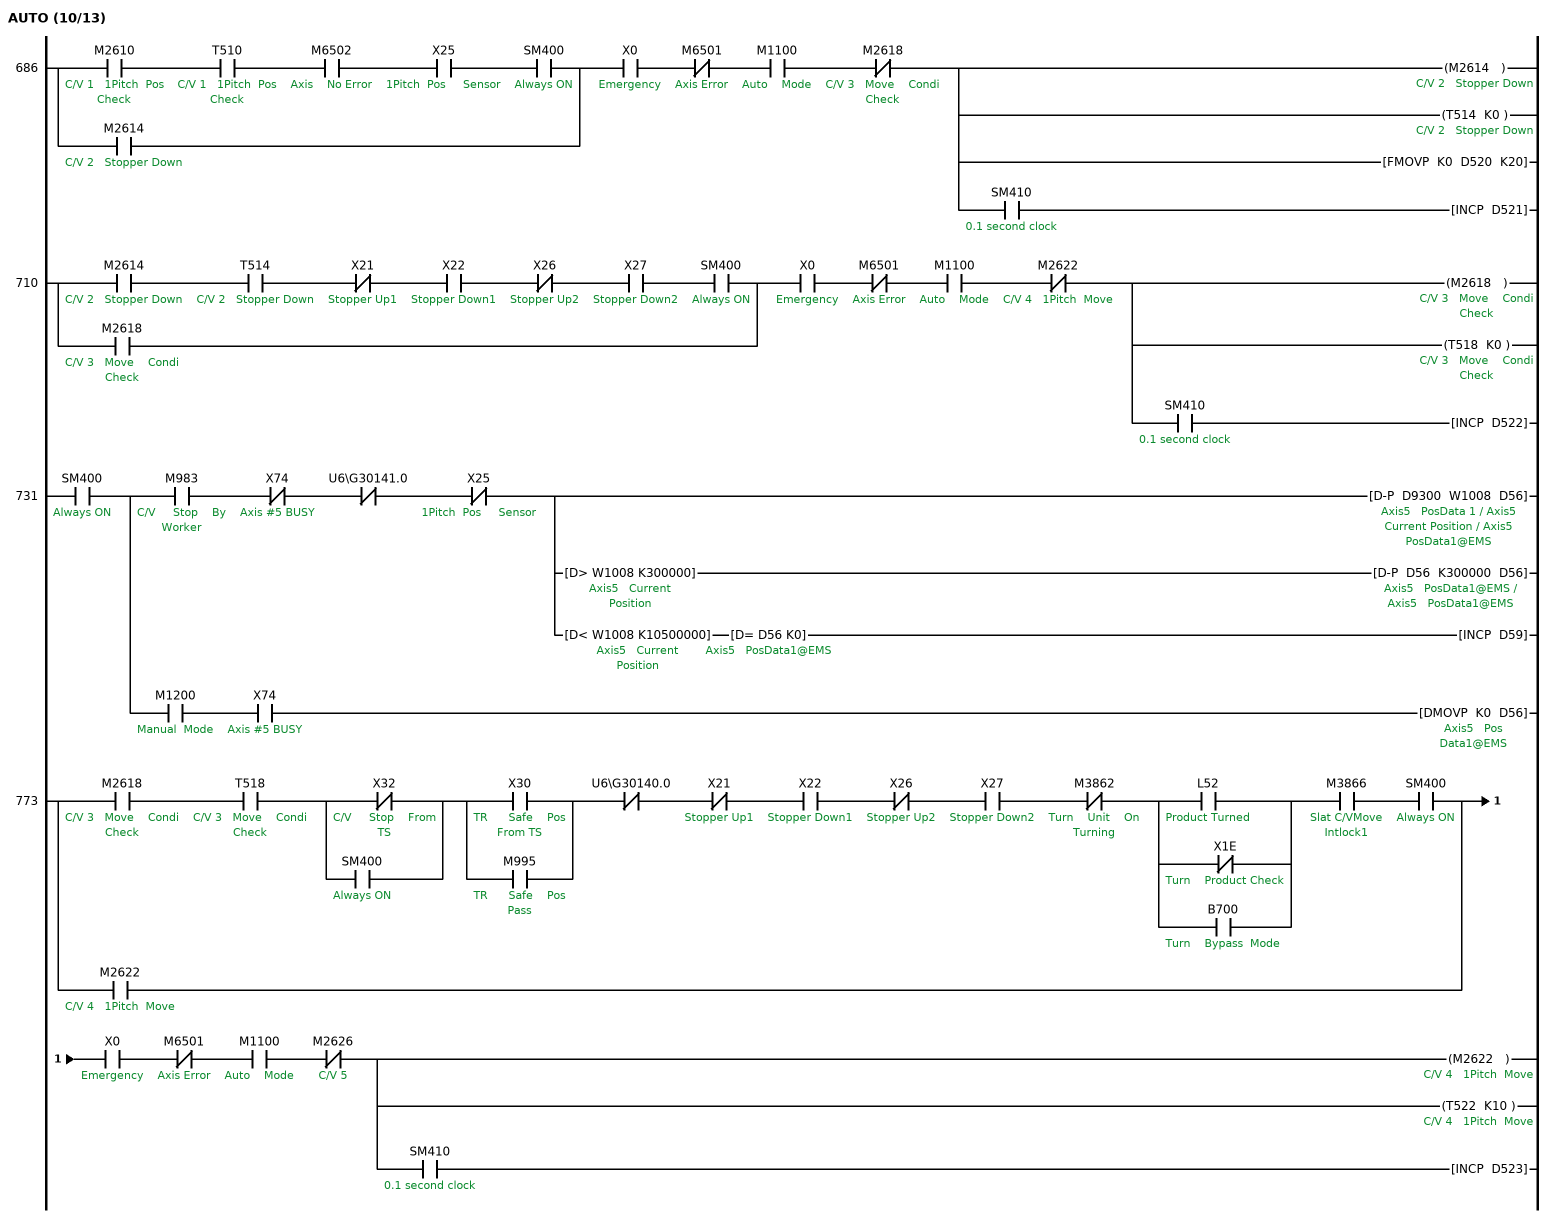
686   LD      M2610  ; C/V 1   1Pitch  Pos     Check
      AND     T510  ; C/V 1   1Pitch  Pos     Check
      AND     M6502  ; Axis    No Error
      AND     X25  ; 1Pitch  Pos     Sensor
      AND     SM400  ; Always ON
      OR      M2614  ; C/V 2   Stopper Down
      AND     X0  ; Emergency
      ANI     M6501  ; Axis Error
      AND     M1100  ; Auto    Mode
      ANI     M2618  ; C/V 3   Move    Condi   Check
      OUT     M2614  ; C/V 2   Stopper Down
      OUT     T514 K0  ; C/V 2   Stopper Down
      FMOVP   K0 D520 K20
      AND     SM410  ; 0.1 second clock
      INCP    D521
710   LD      M2614  ; C/V 2   Stopper Down
      AND     T514  ; C/V 2   Stopper Down
      ANI     X21  ; Stopper Up1
      AND     X22  ; Stopper Down1
      ANI     X26  ; Stopper Up2
      AND     X27  ; Stopper Down2
      AND     SM400  ; Always ON
      OR      M2618  ; C/V 3   Move    Condi   Check
      AND     X0  ; Emergency
      ANI     M6501  ; Axis Error
      AND     M1100  ; Auto    Mode
      ANI     M2622  ; C/V 4   1Pitch  Move
      OUT     M2618  ; C/V 3   Move    Condi   Check
      OUT     T518 K0  ; C/V 3   Move    Condi   Check
      AND     SM410  ; 0.1 second clock
      INCP    D522
731   LD      SM400  ; Always ON
      MPS
      AND     M983  ; C/V     Stop    By      Worker
      ANI     X74  ; Axis #5 BUSY
      ANI     U6\G30141.0
      ANI     X25  ; 1Pitch  Pos     Sensor
      D-P     D9300 W1008 D56  ; Axis5   PosData 1 / Axis5   Current Position / Axis5   PosData1@EMS
      MPS
      ANDD>   W1008 K300000  ; Axis5   Current Position
      D-P     D56 K300000 D56
      MPP
      ANDD<   W1008 K10500000  ; Axis5   Current Position
      ANDD=   D56 K0  ; Axis5   PosData1@EMS
      INCP    D59
      MPP
      AND     M1200  ; Manual  Mode
      AND     X74  ; Axis #5 BUSY
      DMOVP   K0 D56
773   LD      M2618  ; C/V 3   Move    Condi   Check
      AND     T518  ; C/V 3   Move    Condi   Check
      LDI     X32  ; C/V     Stop    From    TS
      OR      SM400  ; Always ON
      ANB
      LD      X30  ; TR      Safe    Pos     From TS
      OR      M995  ; TR      Safe    Pos     Pass
      ANB
      ANI     U6\G30140.0
      ANI     X21  ; Stopper Up1
      AND     X22  ; Stopper Down1
      ANI     X26  ; Stopper Up2
      AND     X27  ; Stopper Down2
      ANI     M3862  ; Turn    Unit    On      Turning
      LD      L52  ; Product Turned
      ORI     X1E  ; Turn    Product Check
      OR      B700  ; Turn    Bypass  Mode
      ANB
      AND     M3866  ; Slat C/VMove    Intlock1
      AND     SM400  ; Always ON
      OR      M2622  ; C/V 4   1Pitch  Move
      AND     X0  ; Emergency
      ANI     M6501  ; Axis Error
      AND     M1100  ; Auto    Mode
      ANI     M2626  ; C/V 5
      OUT     M2622  ; C/V 4   1Pitch  Move
      OUT     T522 K10  ; C/V 4   1Pitch  Move
      AND     SM410  ; 0.1 second clock
      INCP    D523
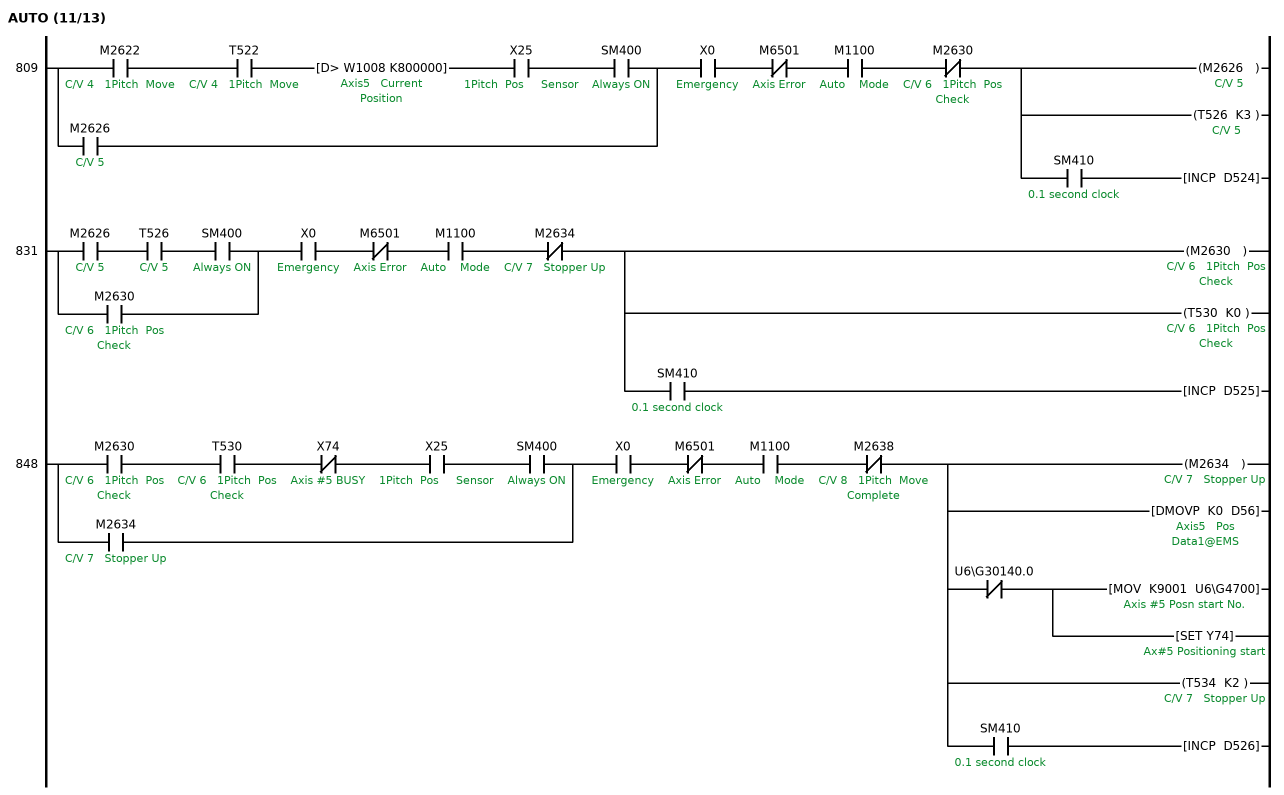
809   LD      M2622  ; C/V 4   1Pitch  Move
      AND     T522  ; C/V 4   1Pitch  Move
      ANDD>   W1008 K800000  ; Axis5   Current Position
      AND     X25  ; 1Pitch  Pos     Sensor
      AND     SM400  ; Always ON
      OR      M2626  ; C/V 5
      AND     X0  ; Emergency
      ANI     M6501  ; Axis Error
      AND     M1100  ; Auto    Mode
      ANI     M2630  ; C/V 6   1Pitch  Pos     Check
      OUT     M2626  ; C/V 5
      OUT     T526 K3  ; C/V 5
      AND     SM410  ; 0.1 second clock
      INCP    D524
831   LD      M2626  ; C/V 5
      AND     T526  ; C/V 5
      AND     SM400  ; Always ON
      OR      M2630  ; C/V 6   1Pitch  Pos     Check
      AND     X0  ; Emergency
      ANI     M6501  ; Axis Error
      AND     M1100  ; Auto    Mode
      ANI     M2634  ; C/V 7   Stopper Up
      OUT     M2630  ; C/V 6   1Pitch  Pos     Check
      OUT     T530 K0  ; C/V 6   1Pitch  Pos     Check
      AND     SM410  ; 0.1 second clock
      INCP    D525
848   LD      M2630  ; C/V 6   1Pitch  Pos     Check
      AND     T530  ; C/V 6   1Pitch  Pos     Check
      ANI     X74  ; Axis #5 BUSY
      AND     X25  ; 1Pitch  Pos     Sensor
      AND     SM400  ; Always ON
      OR      M2634  ; C/V 7   Stopper Up
      AND     X0  ; Emergency
      ANI     M6501  ; Axis Error
      AND     M1100  ; Auto    Mode
      ANI     M2638  ; C/V 8   1Pitch  Move    Complete
      OUT     M2634  ; C/V 7   Stopper Up
      DMOVP   K0 D56
      MPS
      ANI     U6\G30140.0
      MOV     K9001 U6\G4700  ; Axis #5 Posn start No.
      SET     Y74  ; Ax#5 Positioning start
      MPP
      OUT     T534 K2  ; C/V 7   Stopper Up
      AND     SM410  ; 0.1 second clock
      INCP    D526
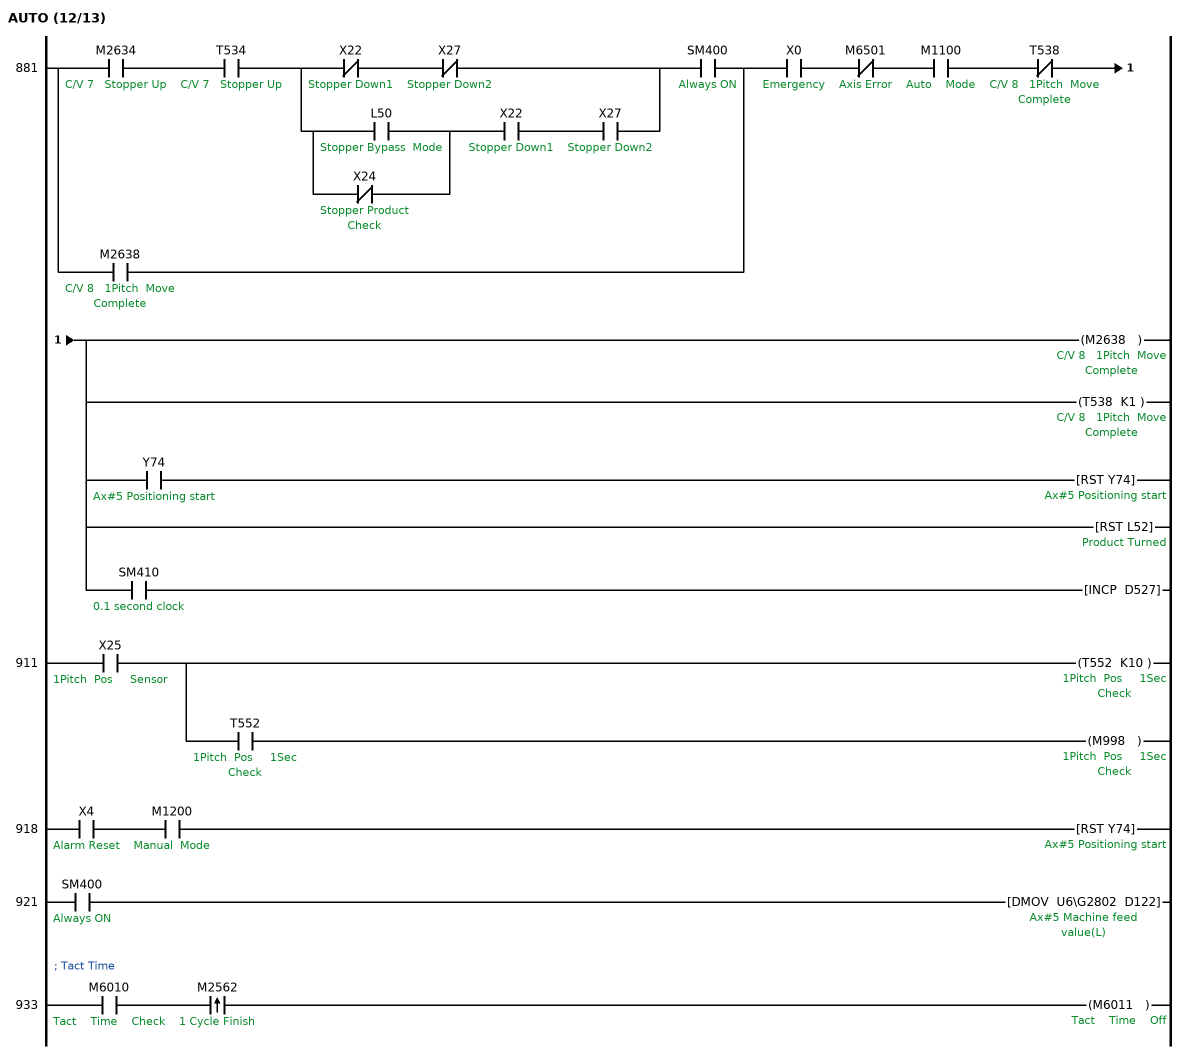
881   LD      M2634  ; C/V 7   Stopper Up
      AND     T534  ; C/V 7   Stopper Up
      LDI     X22  ; Stopper Down1
      ANI     X27  ; Stopper Down2
      LD      L50  ; Stopper Bypass  Mode
      ORI     X24  ; Stopper Product Check
      AND     X22  ; Stopper Down1
      AND     X27  ; Stopper Down2
      ORB
      ANB
      AND     SM400  ; Always ON
      OR      M2638  ; C/V 8   1Pitch  Move    Complete
      AND     X0  ; Emergency
      ANI     M6501  ; Axis Error
      AND     M1100  ; Auto    Mode
      ANI     T538  ; C/V 8   1Pitch  Move    Complete
      OUT     M2638  ; C/V 8   1Pitch  Move    Complete
      OUT     T538 K1  ; C/V 8   1Pitch  Move    Complete
      MPS
      AND     Y74  ; Ax#5 Positioning start
      RST     Y74  ; Ax#5 Positioning start
      MPP
      RST     L52  ; Product Turned
      AND     SM410  ; 0.1 second clock
      INCP    D527
911   LD      X25  ; 1Pitch  Pos     Sensor
      OUT     T552 K10  ; 1Pitch  Pos     1Sec    Check
      AND     T552  ; 1Pitch  Pos     1Sec    Check
      OUT     M998  ; 1Pitch  Pos     1Sec    Check
918   LD      X4  ; Alarm Reset
      AND     M1200  ; Manual  Mode
      RST     Y74  ; Ax#5 Positioning start
921   LD      SM400  ; Always ON
      DMOV    U6\G2802 D122  ; Ax#5 Machine feed value(L)
; Tact Time
933   LD      M6010  ; Tact    Time    Check
      ANDP    M2562  ; 1 Cycle Finish
      OUT     M6011  ; Tact    Time    Off
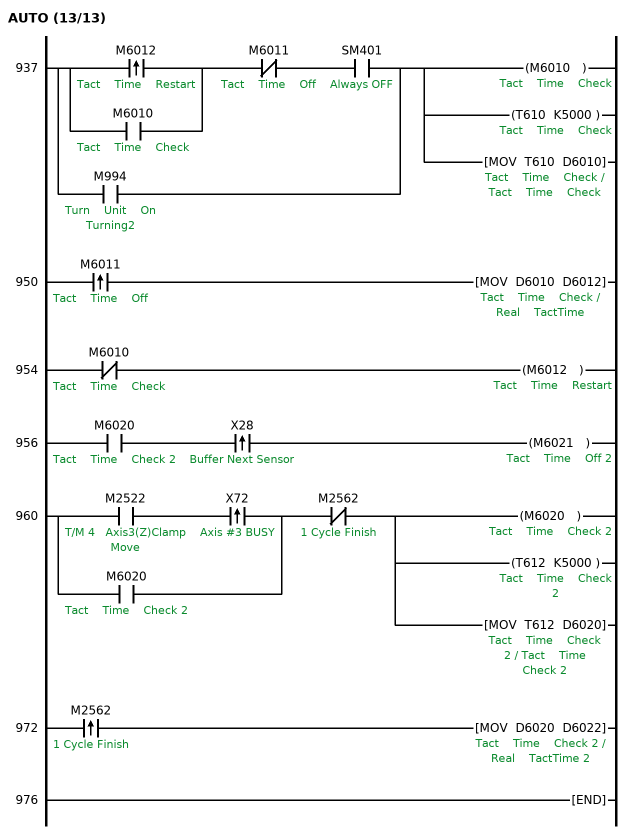
937   LDP     M6012  ; Tact    Time    Restart
      OR      M6010  ; Tact    Time    Check
      ANI     M6011  ; Tact    Time    Off
      AND     SM401  ; Always OFF
      OR      M994  ; Turn    Unit    On      Turning2
      OUT     M6010  ; Tact    Time    Check
      OUT     T610 K5000  ; Tact    Time    Check
      MOV     T610 D6010  ; Tact    Time    Check
950   LDP     M6011  ; Tact    Time    Off
      MOV     D6010 D6012  ; Real    TactTime
954   LDI     M6010  ; Tact    Time    Check
      OUT     M6012  ; Tact    Time    Restart
956   LD      M6020  ; Tact    Time    Check 2
      ANDP    X28  ; Buffer Next Sensor
      OUT     M6021  ; Tact    Time    Off 2
960   LD      M2522  ; T/M 4   Axis3(Z)Clamp   Move
      ANDP    X72  ; Axis #3 BUSY
      OR      M6020  ; Tact    Time    Check 2
      ANI     M2562  ; 1 Cycle Finish
      OUT     M6020  ; Tact    Time    Check 2
      OUT     T612 K5000  ; Tact    Time    Check 2
      MOV     T612 D6020  ; Tact    Time    Check 2
972   LDP     M2562  ; 1 Cycle Finish
      MOV     D6020 D6022  ; Real    TactTime 2
976   END
END_PROGRAM

PROGRAM MANUAL
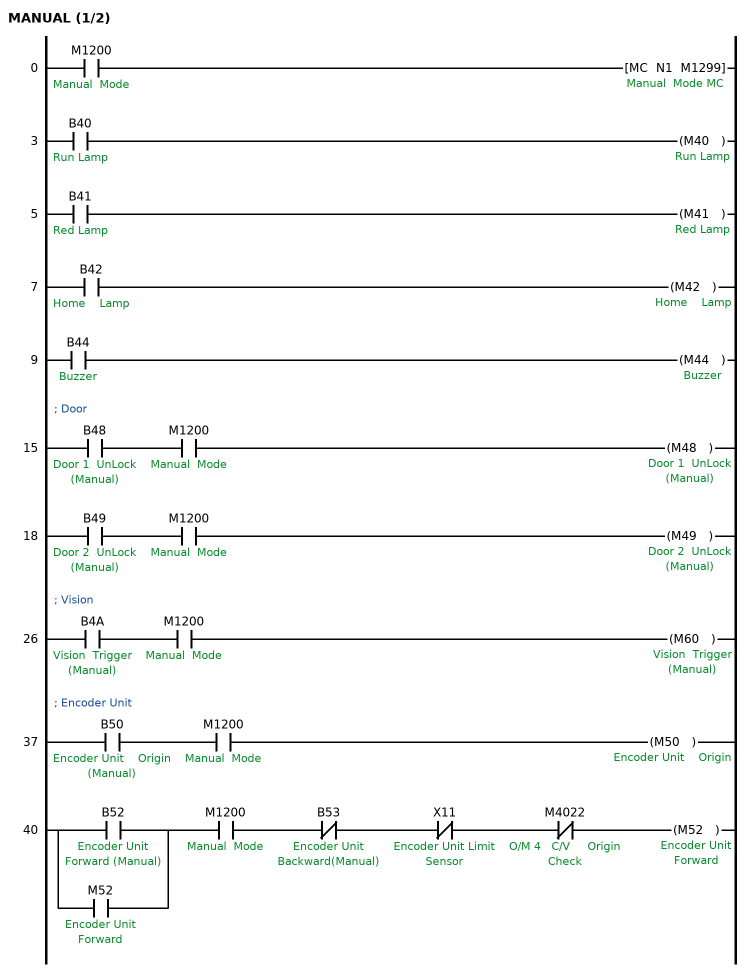
0     LD      M1200  ; Manual  Mode
      MC      N1 M1299  ; Manual  Mode MC
3     LD      B40  ; Run Lamp
      OUT     M40  ; Run Lamp
5     LD      B41  ; Red Lamp
      OUT     M41  ; Red Lamp
7     LD      B42  ; Home    Lamp
      OUT     M42  ; Home    Lamp
9     LD      B44  ; Buzzer
      OUT     M44  ; Buzzer
; Door
15    LD      B48  ; Door 1  UnLock  (Manual)
      AND     M1200  ; Manual  Mode
      OUT     M48  ; Door 1  UnLock  (Manual)
18    LD      B49  ; Door 2  UnLock  (Manual)
      AND     M1200  ; Manual  Mode
      OUT     M49  ; Door 2  UnLock  (Manual)
; Vision
26    LD      B4A  ; Vision  Trigger (Manual)
      AND     M1200  ; Manual  Mode
      OUT     M60  ; Vision  Trigger (Manual)
; Encoder Unit
37    LD      B50  ; Encoder Unit    Origin  (Manual)
      AND     M1200  ; Manual  Mode
      OUT     M50  ; Encoder Unit    Origin
40    LD      B52  ; Encoder Unit    Forward (Manual)
      OR      M52  ; Encoder Unit    Forward
      AND     M1200  ; Manual  Mode
      ANI     B53  ; Encoder Unit    Backward(Manual)
      ANI     X11  ; Encoder Unit Limit Sensor
      ANI     M4022  ; O/M 4   C/V     Origin  Check
      OUT     M52  ; Encoder Unit    Forward
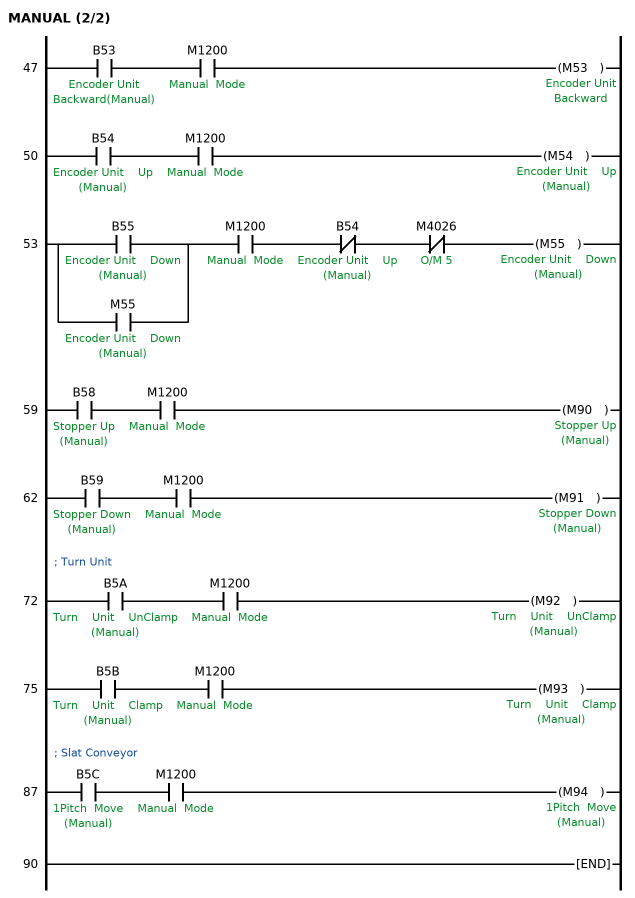
47    LD      B53  ; Encoder Unit    Backward(Manual)
      AND     M1200  ; Manual  Mode
      OUT     M53  ; Encoder Unit    Backward
50    LD      B54  ; Encoder Unit    Up      (Manual)
      AND     M1200  ; Manual  Mode
      OUT     M54  ; Encoder Unit    Up      (Manual)
53    LD      B55  ; Encoder Unit    Down    (Manual)
      OR      M55  ; Encoder Unit    Down    (Manual)
      AND     M1200  ; Manual  Mode
      ANI     B54  ; Encoder Unit    Up      (Manual)
      ANI     M4026  ; O/M 5
      OUT     M55  ; Encoder Unit    Down    (Manual)
59    LD      B58  ; Stopper Up      (Manual)
      AND     M1200  ; Manual  Mode
      OUT     M90  ; Stopper Up      (Manual)
62    LD      B59  ; Stopper Down    (Manual)
      AND     M1200  ; Manual  Mode
      OUT     M91  ; Stopper Down    (Manual)
; Turn Unit
72    LD      B5A  ; Turn    Unit    UnClamp (Manual)
      AND     M1200  ; Manual  Mode
      OUT     M92  ; Turn    Unit    UnClamp (Manual)
75    LD      B5B  ; Turn    Unit    Clamp   (Manual)
      AND     M1200  ; Manual  Mode
      OUT     M93  ; Turn    Unit    Clamp   (Manual)
; Slat Conveyor
87    LD      B5C  ; 1Pitch  Move    (Manual)
      AND     M1200  ; Manual  Mode
      OUT     M94  ; 1Pitch  Move    (Manual)
90    END
END_PROGRAM

PROGRAM ORIGIN
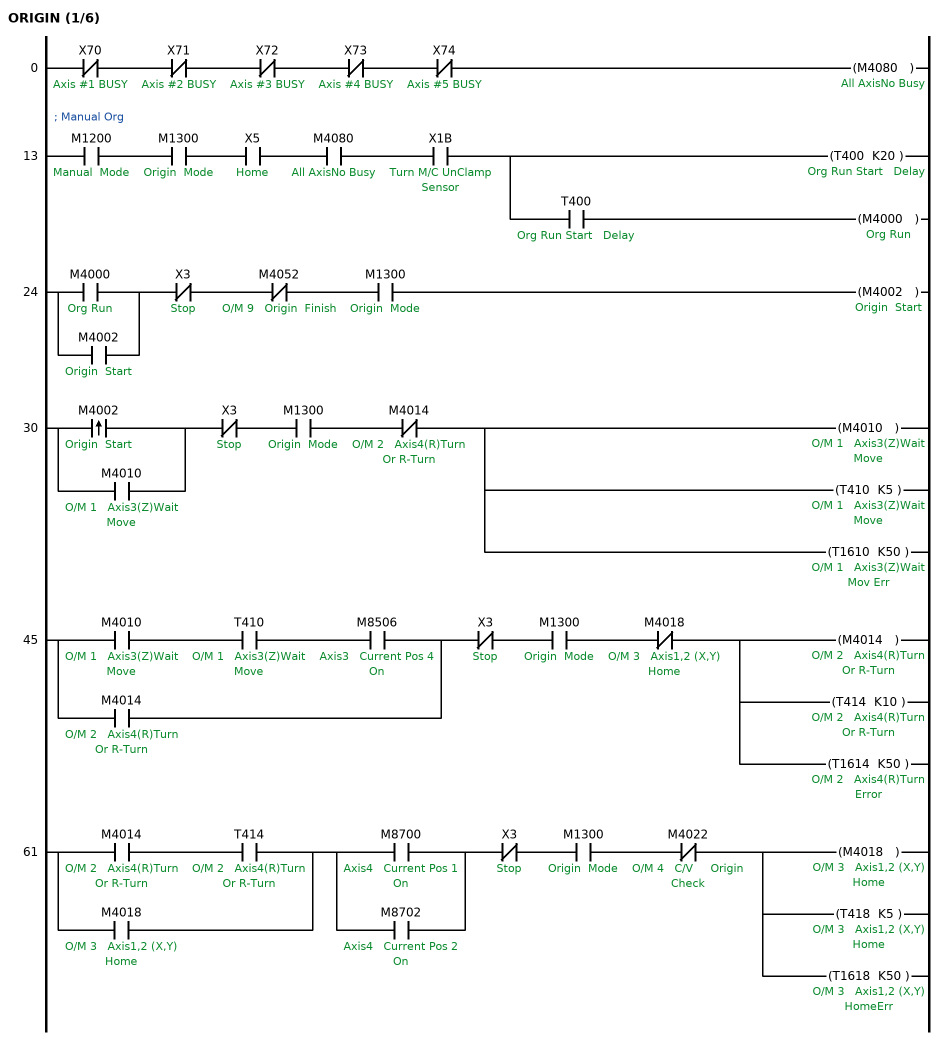
0     LDI     X70  ; Axis #1 BUSY
      ANI     X71  ; Axis #2 BUSY
      ANI     X72  ; Axis #3 BUSY
      ANI     X73  ; Axis #4 BUSY
      ANI     X74  ; Axis #5 BUSY
      OUT     M4080  ; All AxisNo Busy
; Manual Org
13    LD      M1200  ; Manual  Mode
      AND     M1300  ; Origin  Mode
      AND     X5  ; Home
      AND     M4080  ; All AxisNo Busy
      AND     X1B  ; Turn M/C UnClamp Sensor
      OUT     T400 K20  ; Org Run Start   Delay
      AND     T400  ; Org Run Start   Delay
      OUT     M4000  ; Org Run
24    LD      M4000  ; Org Run
      OR      M4002  ; Origin  Start
      ANI     X3  ; Stop
      ANI     M4052  ; O/M 9   Origin  Finish
      AND     M1300  ; Origin  Mode
      OUT     M4002  ; Origin  Start
30    LDP     M4002  ; Origin  Start
      OR      M4010  ; O/M 1   Axis3(Z)Wait    Move
      ANI     X3  ; Stop
      AND     M1300  ; Origin  Mode
      ANI     M4014  ; O/M 2   Axis4(R)Turn Or R-Turn
      OUT     M4010  ; O/M 1   Axis3(Z)Wait    Move
      OUT     T410 K5  ; O/M 1   Axis3(Z)Wait    Move
      OUT     T1610 K50  ; O/M 1   Axis3(Z)Wait    Mov Err
45    LD      M4010  ; O/M 1   Axis3(Z)Wait    Move
      AND     T410  ; O/M 1   Axis3(Z)Wait    Move
      AND     M8506  ; Axis3   Current Pos 4 On
      OR      M4014  ; O/M 2   Axis4(R)Turn Or R-Turn
      ANI     X3  ; Stop
      AND     M1300  ; Origin  Mode
      ANI     M4018  ; O/M 3   Axis1,2 (X,Y)   Home
      OUT     M4014  ; O/M 2   Axis4(R)Turn Or R-Turn
      OUT     T414 K10  ; O/M 2   Axis4(R)Turn Or R-Turn
      OUT     T1614 K50  ; O/M 2   Axis4(R)Turn    Error
61    LD      M4014  ; O/M 2   Axis4(R)Turn Or R-Turn
      AND     T414  ; O/M 2   Axis4(R)Turn Or R-Turn
      OR      M4018  ; O/M 3   Axis1,2 (X,Y)   Home
      LD      M8700  ; Axis4   Current Pos 1 On
      OR      M8702  ; Axis4   Current Pos 2 On
      ANB
      ANI     X3  ; Stop
      AND     M1300  ; Origin  Mode
      ANI     M4022  ; O/M 4   C/V     Origin  Check
      OUT     M4018  ; O/M 3   Axis1,2 (X,Y)   Home
      OUT     T418 K5  ; O/M 3   Axis1,2 (X,Y)   Home
      OUT     T1618 K50  ; O/M 3   Axis1,2 (X,Y)   HomeErr
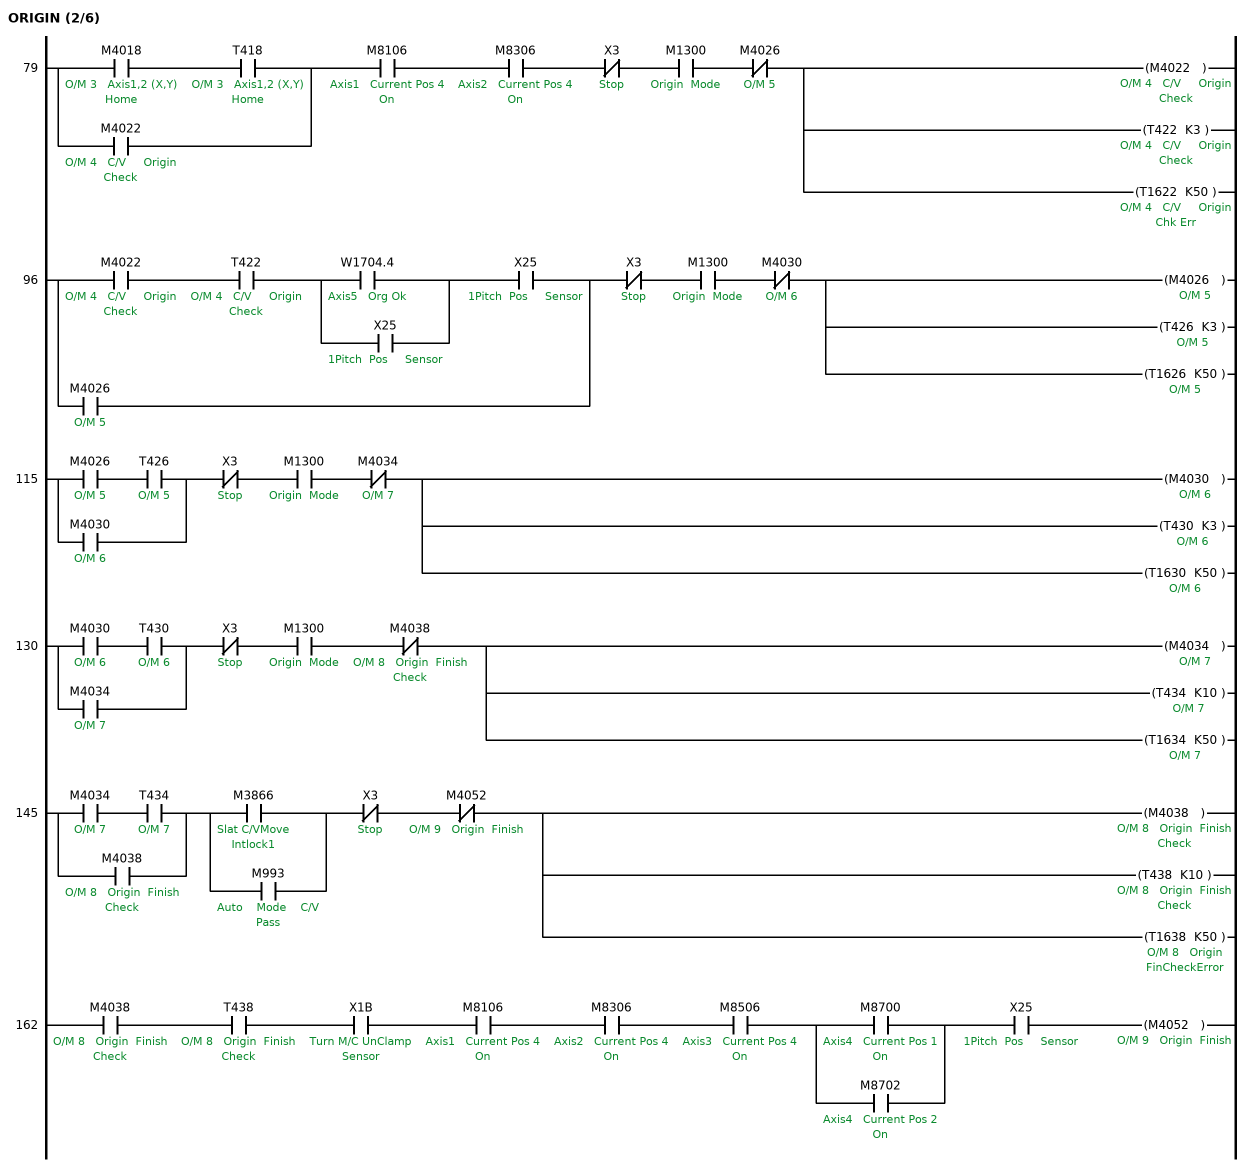
79    LD      M4018  ; O/M 3   Axis1,2 (X,Y)   Home
      AND     T418  ; O/M 3   Axis1,2 (X,Y)   Home
      OR      M4022  ; O/M 4   C/V     Origin  Check
      AND     M8106  ; Axis1   Current Pos 4 On
      AND     M8306  ; Axis2   Current Pos 4 On
      ANI     X3  ; Stop
      AND     M1300  ; Origin  Mode
      ANI     M4026  ; O/M 5
      OUT     M4022  ; O/M 4   C/V     Origin  Check
      OUT     T422 K3  ; O/M 4   C/V     Origin  Check
      OUT     T1622 K50  ; O/M 4   C/V     Origin  Chk Err
96    LD      M4022  ; O/M 4   C/V     Origin  Check
      AND     T422  ; O/M 4   C/V     Origin  Check
      LD      W1704.4  ; Axis5   Org Ok
      OR      X25  ; 1Pitch  Pos     Sensor
      ANB
      AND     X25  ; 1Pitch  Pos     Sensor
      OR      M4026  ; O/M 5
      ANI     X3  ; Stop
      AND     M1300  ; Origin  Mode
      ANI     M4030  ; O/M 6
      OUT     M4026  ; O/M 5
      OUT     T426 K3  ; O/M 5
      OUT     T1626 K50  ; O/M 5
115   LD      M4026  ; O/M 5
      AND     T426  ; O/M 5
      OR      M4030  ; O/M 6
      ANI     X3  ; Stop
      AND     M1300  ; Origin  Mode
      ANI     M4034  ; O/M 7
      OUT     M4030  ; O/M 6
      OUT     T430 K3  ; O/M 6
      OUT     T1630 K50  ; O/M 6
130   LD      M4030  ; O/M 6
      AND     T430  ; O/M 6
      OR      M4034  ; O/M 7
      ANI     X3  ; Stop
      AND     M1300  ; Origin  Mode
      ANI     M4038  ; O/M 8   Origin  Finish  Check
      OUT     M4034  ; O/M 7
      OUT     T434 K10  ; O/M 7
      OUT     T1634 K50  ; O/M 7
145   LD      M4034  ; O/M 7
      AND     T434  ; O/M 7
      OR      M4038  ; O/M 8   Origin  Finish  Check
      LD      M3866  ; Slat C/VMove    Intlock1
      OR      M993  ; Auto    Mode    C/V     Pass
      ANB
      ANI     X3  ; Stop
      ANI     M4052  ; O/M 9   Origin  Finish
      OUT     M4038  ; O/M 8   Origin  Finish  Check
      OUT     T438 K10  ; O/M 8   Origin  Finish  Check
      OUT     T1638 K50  ; O/M 8   Origin  FinCheckError
162   LD      M4038  ; O/M 8   Origin  Finish  Check
      AND     T438  ; O/M 8   Origin  Finish  Check
      AND     X1B  ; Turn M/C UnClamp Sensor
      AND     M8106  ; Axis1   Current Pos 4 On
      AND     M8306  ; Axis2   Current Pos 4 On
      AND     M8506  ; Axis3   Current Pos 4 On
      LD      M8700  ; Axis4   Current Pos 1 On
      OR      M8702  ; Axis4   Current Pos 2 On
      ANB
      AND     X25  ; 1Pitch  Pos     Sensor
      OUT     M4052  ; O/M 9   Origin  Finish
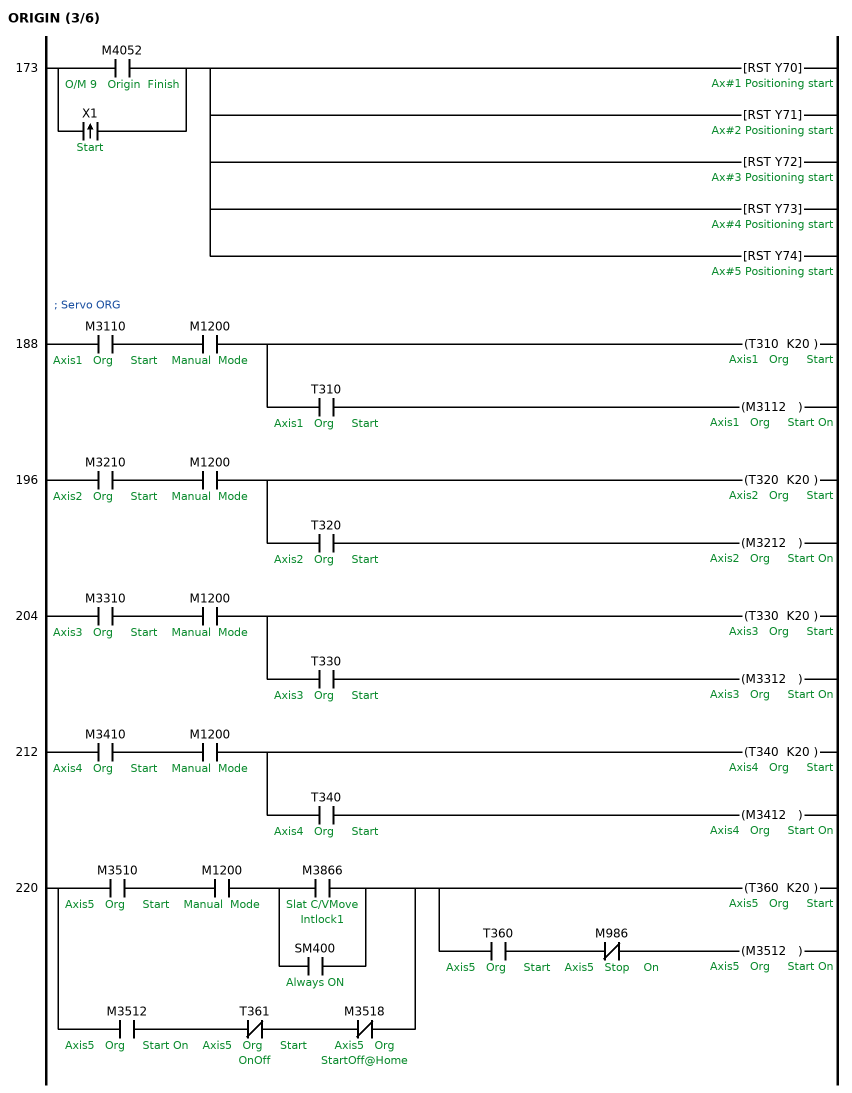
173   LD      M4052  ; O/M 9   Origin  Finish
      ORP     X1  ; Start
      RST     Y70  ; Ax#1 Positioning start
      RST     Y71  ; Ax#2 Positioning start
      RST     Y72  ; Ax#3 Positioning start
      RST     Y73  ; Ax#4 Positioning start
      RST     Y74  ; Ax#5 Positioning start
; Servo ORG
188   LD      M3110  ; Axis1   Org     Start
      AND     M1200  ; Manual  Mode
      OUT     T310 K20  ; Axis1   Org     Start
      AND     T310  ; Axis1   Org     Start
      OUT     M3112  ; Axis1   Org     Start On
196   LD      M3210  ; Axis2   Org     Start
      AND     M1200  ; Manual  Mode
      OUT     T320 K20  ; Axis2   Org     Start
      AND     T320  ; Axis2   Org     Start
      OUT     M3212  ; Axis2   Org     Start On
204   LD      M3310  ; Axis3   Org     Start
      AND     M1200  ; Manual  Mode
      OUT     T330 K20  ; Axis3   Org     Start
      AND     T330  ; Axis3   Org     Start
      OUT     M3312  ; Axis3   Org     Start On
212   LD      M3410  ; Axis4   Org     Start
      AND     M1200  ; Manual  Mode
      OUT     T340 K20  ; Axis4   Org     Start
      AND     T340  ; Axis4   Org     Start
      OUT     M3412  ; Axis4   Org     Start On
220   LD      M3510  ; Axis5   Org     Start
      AND     M1200  ; Manual  Mode
      LD      M3866  ; Slat C/VMove    Intlock1
      OR      SM400  ; Always ON
      ANB
      LD      M3512  ; Axis5   Org     Start On
      ANI     T361  ; Axis5   Org     Start OnOff
      ANI     M3518  ; Axis5   Org     StartOff@Home
      ORB
      OUT     T360 K20  ; Axis5   Org     Start
      AND     T360  ; Axis5   Org     Start
      ANI     M986  ; Axis5   Stop    On
      OUT     M3512  ; Axis5   Org     Start On
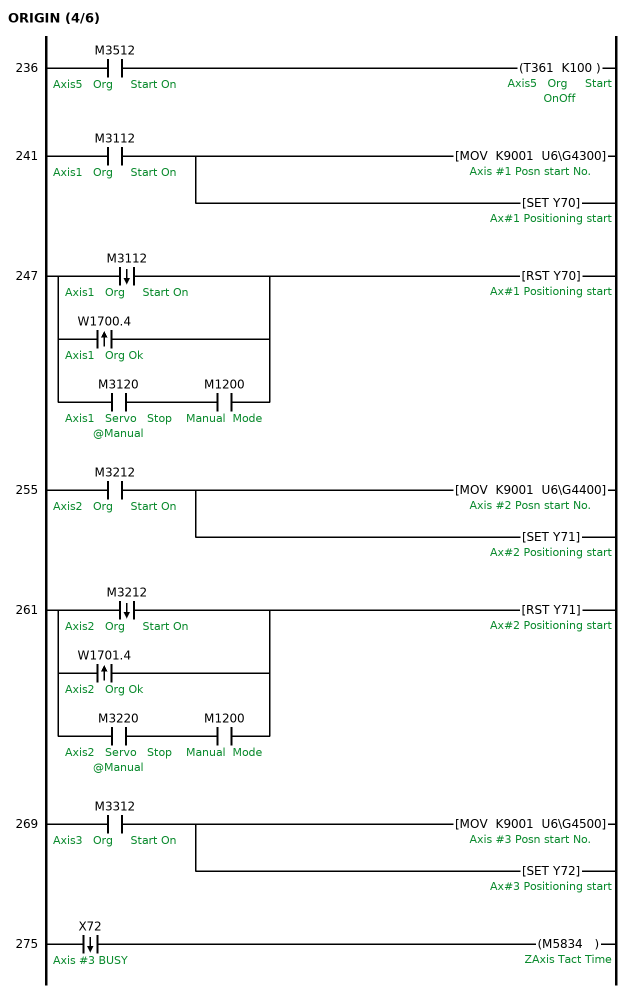
236   LD      M3512  ; Axis5   Org     Start On
      OUT     T361 K100  ; Axis5   Org     Start OnOff
241   LD      M3112  ; Axis1   Org     Start On
      MOV     K9001 U6\G4300  ; Axis #1 Posn start No.
      SET     Y70  ; Ax#1 Positioning start
247   LDF     M3112  ; Axis1   Org     Start On
      ORP     W1700.4  ; Axis1   Org Ok
      LD      M3120  ; Axis1   Servo   Stop    @Manual
      AND     M1200  ; Manual  Mode
      ORB
      RST     Y70  ; Ax#1 Positioning start
255   LD      M3212  ; Axis2   Org     Start On
      MOV     K9001 U6\G4400  ; Axis #2 Posn start No.
      SET     Y71  ; Ax#2 Positioning start
261   LDF     M3212  ; Axis2   Org     Start On
      ORP     W1701.4  ; Axis2   Org Ok
      LD      M3220  ; Axis2   Servo   Stop    @Manual
      AND     M1200  ; Manual  Mode
      ORB
      RST     Y71  ; Ax#2 Positioning start
269   LD      M3312  ; Axis3   Org     Start On
      MOV     K9001 U6\G4500  ; Axis #3 Posn start No.
      SET     Y72  ; Ax#3 Positioning start
275   LDF     X72  ; Axis #3 BUSY
      OUT     M5834  ; ZAxis Tact Time
